  (* -------------------------------------------------------------
    Load-Error 							
  --------------------------------------------------------------*)
  JAM_ERROR                                 := 0180, // Jam Detected - Remove TU before restart 
  POSITION_OCCUPIED_AFTER_HANDOVER          := 0181, // Position occupied after transmission 
  POSITION_OCCUPIED_BEFORE_TAKEOVER         := 0182, // Position occupied before pickup 
  POSITION_NOT_CORRECT_OCCUPIED             := 0183, // Position is not correctly occupied 
  LOAD_CONTROL                              := 0184, // Check load for overhang 
  POSITION_LANE_FULL                        := 0185, // Position/Lane is full, remove some TU's 
  TRANSFER_ERROR                            := 0186, // Error during transfer
  LOAD_TOO_HIGH                             := 0187, // Load is too high
  LOAD_TOO_HEAVY                            := 0188, // Load is too heavy


  (* -------------------------------------------------------------
    Errors Drives						
  --------------------------------------------------------------*)
  DRIVE_ERROR                               := 0200, // Drive error 
  DRIVE_WARNING                             := 0201, // Drive warning 


  (*-------------------------------------------------------------
    Errors Scanners						
  --------------------------------------------------------------*)
  SCANNER_NO_READ                           := 0220, // Scanner could not read the label 
  SCANNER_CONTINOUS_NO_READ                 := 0221, // Continuous no reading 
  SCANNER_NO_DATA_RECEIVED                  := 0222, // No data received from scanner 
  SCANNER_NO_HANDSHAKE                      := 0223, // No handshake signal from scanner received 


  (* -------------------------------------------------------------
    Misc      
  --------------------------------------------------------------*)
  INIT_NOT_POSSIBLE                         := 0300, // Initialization was not possible
  START_NOT_POSSIBLE                        := 0301, // Starting not possible
  POSITIONING_ERROR                         := 0302, // Positioning error 
  INCORRECT_POSITION                        := 0303, // Actual position is not correct 
  BELT_BROKEN                               := 0304, // Belt is broken 
  DEVICE_ERROR                              := 0305, // Device error
  DEVICE_OFFLINE                            := 0306, // device is offline e.g. printer, scanner 
  WATCHDOG_ERROR                            := 0307, // Watchdog error 
  FILE_SYSTEM_ERROR                         := 0308, // Error during deleting file 
  DOOR_ERROR                                := 0309, // Maintenance door is open error 
  WRONG_MODE                                := 0310, // Manual mode is not active for performing manual movement 
  NOT_SUPPORTED                             := 0311, // Not supported message


  (* -------------------------------------------------------------
    Software errors       
  --------------------------------------------------------------*)
  CONFIGURATION_ERROR                       := 0900, // Configuration error 
  SOFTWARE_ERROR                            := 0901  // General software error 
);
END_TYPE

// ---- 20_Product/10_BCF/11_Conv/10_Base/01_DUTs/E_EtherCAT_MasterError.TcDUT
TYPE E_EtherCAT_MasterError :
(**************************************************************************************
 * 	Application		:	BoxControl Framework
 *	Revision		:	$Revision: 404529 $
 *	Revision date	:	$Date: 2018-04-23 08:21:38 +0200 (Mo., 23 Apr 2018) $
 *	Last changed by	:	$Author: b7bolm $
 *	URL				:	$URL: http://almscdc.swisslog.com/repo/SWPD/Development/BoxControlFramework/20_Release/trunk/01_Software/BCF/BCF/JumpStart/20_Product/10_App/10_Base/10_Lib/10_Conv/01_DUTs/E_EtherCAT_MasterError.TcDUT $
 *
 *	Purpose			:	EtherCAT master error
 *
 * ------------------------------------------------------------------------------------
 *	Copyright Swisslog [IP AG], Switzerland. All rights reserved.
 * 
 * ------------------------------------------------------------------------------------
 *	
 * 	Revision History: 
 *
 * 	VERSION			DATE			INITIALS			DESCRIPTION
 *	0.1				01.01.2001		swl					Example
 *
 **************************************************************************************)
(
	ETHERCAT_MASTER_NO_ERROR		:= 16#0000, // No error 
	LINK_ERROR 						:= 16#0001, // Link error  
	IO_LOCKED_AFTER_LINK_ERR		:= 16#0002, // I/O locked after link error (I/O reset required) 
	LINK_ERROR_REDUNDANCY_ADAPTER	:= 16#0004, // Link error (redundancy adapter) 
	MISSING_ONE_FRAME				:= 16#0008, // Missing one frame (redundancy mode) 
	OUT_OF_SEND_RESSOURCES			:= 16#0010, // Out OF send resources (I/O reset required) 
	WATCHDOG_TRIGGERED				:= 16#0020, // Watchdog triggered 
	ETHERNET_DRV_NOT_FOUND			:= 16#0040, // Ethernet driver (miniport) NOT found 
	IO_RESET_ACTIVE					:= 16#0080, // I/O reset active
	ONE_DEVICE_IN_INIT				:= 16#0100, // AT least one device in 'INIT' state 
	ONE_DEVICE_IN_PRE_OP			:= 16#0200, // AT least one device in 'PRE-OP' state 
	ONE_DEVICE_IN_SAFE_OP			:= 16#0400, // AT least one device in 'SAFE-OP' state 
	ONE_DEVICE_IN_ERROR				:= 16#0800, // AT least one device indicates an error state 
	DC_NOT_IN_SYNC					:= 16#1000  // DC NOT in sync 
);
END_TYPE

// ---- 20_Product/10_BCF/11_Conv/10_Base/01_DUTs/ST_ControlRequest.TcDUT
TYPE ST_ControlRequest :
(**************************************************************************************
 * 	Application		:	BoxControl Framework
 *	Revision		:	$Revision: 404529 $
 *	Revision date	:	$Date: 2018-04-23 08:21:38 +0200 (Mo., 23 Apr 2018) $
 *	Last changed by	:	$Author: b7bolm $
 *	URL				:	$URL: http://almscdc.swisslog.com/repo/SWPD/Development/BoxControlFramework/20_Release/trunk/01_Software/BCF/BCF/JumpStart/20_Product/10_App/10_Base/10_Lib/10_Conv/01_DUTs/ST_ControlRequest.TcDUT $
 *
 *	Purpose			:	Control request consists of a control code and value. These 
 *						values are normaly set by an ITC message.
 *
 * ------------------------------------------------------------------------------------
 *	Copyright Swisslog [IP AG], Switzerland. All rights reserved.
 * 
 * ------------------------------------------------------------------------------------
 *	
 * 	Revision History: 
 *
 * 	VERSION			DATE			INITIALS			DESCRIPTION
 *	0.1				01.01.2001		swl					Example
 *
 **************************************************************************************)
STRUCT
	ControlCode			: INT; // Control code from the control telegram 
	ControlValue		: INT; // Control value from the control telegram 
END_STRUCT
END_TYPE

// ---- 20_Product/10_BCF/11_Conv/10_Base/01_DUTs/ST_DataSet.TcDUT
TYPE ST_DataSet :
(**************************************************************************************
 * 	Application		:	BoxControl Framework
 *	Revision		:	$Revision: 411223 $
 *	Revision date	:	$Date: 2018-07-27 11:40:44 +0200 (Fr., 27 Jul 2018) $
 *	Last changed by	:	$Author: b7bolm $
 *	URL				:	$URL: http://almscdc.swisslog.com/repo/SWPD/Development/BoxControlFramework/20_Release/trunk/01_Software/BCF/BCF/JumpStart/20_Product/10_App/10_Base/10_Lib/10_Conv/01_DUTs/ST_DataSet.TcDUT $
 *
 *	Purpose			:	TU Data - Data set
 *
 * ------------------------------------------------------------------------------------
 *	Copyright Swisslog [IP AG], Switzerland. All rights reserved.
 * 
 * ------------------------------------------------------------------------------------
 *	
 * 	Revision History: 
 *
 * 	VERSION			DATE			INITIALS			DESCRIPTION
 *	0.1				01.01.2001		swl					Example
 *
 **************************************************************************************)
STRUCT
	DataPresent		: BOOL; // Data present 
	JobPresent		: BOOL; // Transfer order 
	TU_Type			: INT; // Type of transport unit 
	IO_Data			: INT; // Project specific data 
	Sequence		: ULINT; // 19 digit global sequence identifier
	SubSequence		: DINT; // 9 digit position in the sequence
	SequenceSize	: DINT; // 9 digit number of TU's in the sequence
	GroupID			: ULINT; // 19 digit global group identifier 
	GroupSize		: DINT; // 9 digit number of TU's in the group ID
	DestinationSlot	: INT; // 3 digit logical sub destination of destination
	NumberOfDest	: INT; // Number of destinations 
	Dimension		: ST_Dimension; // Dimensions
	Orientation		: STRING;	
	LowerLimit		: DINT; // Lower limit 
	UpperLimit		: DINT; // Upper limit
	TU_Parameter	: INT; // TU Parameter
	CheckpointID	: STRING(5); // Checkpoint ID
	HaltSequencing	: BOOL; // Sequencing information is temporally not valid
END_STRUCT
END_TYPE

// ---- 20_Product/10_BCF/11_Conv/10_Base/01_DUTs/ST_DataSetEmulation.TcDUT
TYPE ST_DataSetEmulation :
(**************************************************************************************
 * 	Application		:	BoxControl Framework
 *	Revision		:	$Revision: 404529 $
 *	Revision date	:	$Date: 2018-04-23 08:21:38 +0200 (Mo., 23 Apr 2018) $
 *	Last changed by	:	$Author: b7bolm $
 *	URL				:	$URL: http://almscdc.swisslog.com/repo/SWPD/Development/BoxControlFramework/20_Release/trunk/01_Software/BCF/BCF/JumpStart/20_Product/11_Emu/10_Base/10_Lib/10_Conv/01_DUTs/ST_DataSetEmulation.TcDUT $
 *
 *	Purpose			:	TU Data - Data set - Emulation
 *
 * ------------------------------------------------------------------------------------
 *	Copyright Swisslog [IP AG], Switzerland. All rights reserved.
 * 
 * ------------------------------------------------------------------------------------
 *	
 * 	Revision History: 
 *
 * 	VERSION			DATE			INITIALS			DESCRIPTION
 *	0.1				01.01.2001		swl					Example
 *
 **************************************************************************************)
STRUCT
	DataPresent		: BOOL; // Data present
	LongSideLeading : BOOL; // TU runs long side leading
	NestedIndex		: DINT; // Index of nested data set
	ParentIndex		: DINT; // Index of parent in view of nested
 	Dimension		: ST_Dimension; // Dimensions
END_STRUCT
END_TYPE

// ---- 20_Product/10_BCF/11_Conv/10_Base/01_DUTs/ST_Dimension.TcDUT
TYPE ST_Dimension :
(**************************************************************************************
 * 	Application		:	BoxControl Framework
 *	Revision		:	$Revision: 404529 $
 *	Revision date	:	$Date: 2018-04-23 08:21:38 +0200 (Mo., 23 Apr 2018) $
 *	Last changed by	:	$Author: b7bolm $
 *	URL				:	$URL: http://almscdc.swisslog.com/repo/SWPD/Development/BoxControlFramework/20_Release/trunk/01_Software/BCF/BCF/JumpStart/20_Product/10_App/10_Base/10_Lib/10_Conv/01_DUTs/ST_Dimension.TcDUT $
 *
 *	Purpose			:	TU Data - Dimension
 *
 * ------------------------------------------------------------------------------------
 *	Copyright Swisslog [IP AG], Switzerland. All rights reserved.
 * 
 * ------------------------------------------------------------------------------------
 *	
 * 	Revision History: 
 *
 * 	VERSION			DATE			INITIALS			DESCRIPTION
 *	0.1				01.01.2001		swl					Example
 *
 **************************************************************************************)
STRUCT
	Length		: INT; // Length
	Width		: INT; // Width
	Height		: INT; // Height
	Weight		: DINT; // Weight
END_STRUCT
END_TYPE

// ---- 20_Product/10_BCF/11_Conv/10_Base/01_DUTs/ST_ElementRegistryConv.TcDUT
TYPE ST_ElementRegistryConv :
(**************************************************************************************
 * 	Application		:	BoxControl Framework
 *	Revision		:	$Revision: 404529 $
 *	Revision date	:	$Date: 2018-04-23 08:21:38 +0200 (Mo., 23 Apr 2018) $
 *	Last changed by	:	$Author: b7bolm $
 *	URL				:	$URL: http://almscdc.swisslog.com/repo/SWPD/Development/BoxControlFramework/20_Release/trunk/01_Software/BCF/BCF/JumpStart/20_Product/10_App/10_Base/10_Lib/10_Conv/01_DUTs/ST_ElementRegistryConv.TcDUT $
 *
 *	Purpose			:	Element registration structure.
 *
 * ------------------------------------------------------------------------------------
 *	Copyright Swisslog [IP AG], Switzerland. All rights reserved.
 * 
 * ------------------------------------------------------------------------------------
 *	
 * 	Revision History: 
 *
 * 	VERSION			DATE			INITIALS			DESCRIPTION
 *	0.1				01.01.2001		swl					Example
 *
 **************************************************************************************)
STRUCT
	Enable				: BOOL; // Element enabled 
	ElementName			: STRING(System.NAME_LENGTH); // Name as string
	eElementNumber		: E_ElementNumber; // Element number 
	eElementType		: E_ElementType; // Element type
	rElementData		: REFERENCE TO ST_ElementData; 
	rElementInterface 	: REFERENCE TO ST_ElementInterface;
	rSettingsElement	: REFERENCE TO ST_CFG_Element;
	rElement			: REFERENCE TO FB_ElementConv; // Reference to Element 
	HashCode			: UDINT; // HashCode
END_STRUCT
END_TYPE

// ---- 20_Product/10_BCF/11_Conv/10_Base/01_DUTs/ST_ElementRegistryConvEmulation.TcDUT
TYPE ST_ElementRegistryConvEmulation :
(**************************************************************************************
 * 	Application		:	BoxControl Framework
 *	Revision		:	$Revision: 404529 $
 *	Revision date	:	$Date: 2018-04-23 08:21:38 +0200 (Mo., 23 Apr 2018) $
 *	Last changed by	:	$Author: b7bolm $
 *	URL				:	$URL: http://almscdc.swisslog.com/repo/SWPD/Development/BoxControlFramework/20_Release/trunk/01_Software/BCF/BCF/JumpStart/20_Product/11_Emu/10_Base/10_Lib/10_Conv/01_DUTs/ST_ElementRegistryConvEmulation.TcDUT $
 *
 *	Purpose			:	Element registration structure - Emulation.
 *
 * ------------------------------------------------------------------------------------
 *	Copyright Swisslog [IP AG], Switzerland. All rights reserved.
 * 
 * ------------------------------------------------------------------------------------
 *	
 * 	Revision History: 
 *
 * 	VERSION			DATE			INITIALS			DESCRIPTION
 *	0.1				01.01.2001		swl					Example
 *
 **************************************************************************************)
STRUCT
	rElement			: REFERENCE TO FB_ElementConvEmulation; // Element object reference
END_STRUCT
END_TYPE

// ---- 20_Product/10_BCF/11_Conv/10_Base/01_DUTs/ST_ErrorDataSet.TcDUT
TYPE ST_ErrorDataSet :
(**************************************************************************************
 * 	Application		:	BoxControl Framework
 *	Revision		:	$Revision: 404529 $
 *	Revision date	:	$Date: 2018-04-23 08:21:38 +0200 (Mo., 23 Apr 2018) $
 *	Last changed by	:	$Author: b7bolm $
 *	URL				:	$URL: http://almscdc.swisslog.com/repo/SWPD/Development/BoxControlFramework/20_Release/trunk/01_Software/BCF/BCF/JumpStart/20_Product/10_App/10_Base/10_Lib/10_Conv/01_DUTs/ST_ErrorDataSet.TcDUT $
 *
 *	Purpose			:	Error data set
 *
 * ------------------------------------------------------------------------------------
 *	Copyright Swisslog [IP AG], Switzerland. All rights reserved.
 * 
 * ------------------------------------------------------------------------------------
 *	
 * 	Revision History: 
 *
 * 	VERSION			DATE			INITIALS			DESCRIPTION
 *	0.1				01.01.2001		swl					Example
 *
 **************************************************************************************)
STRUCT
	ErrorType		: E_ErrorType;	// Type of error 
	ErrorCode		: U_ErrorCode; // Type casting for error code by product or framework errors 
	ErrorParam		: STRING(System.ERROR_PARAM_STRINGLENGTH); // Error parameter 
	ResetError		: BOOL; // Command to reset error 
END_STRUCT
END_TYPE

// ---- 20_Product/10_BCF/11_Conv/10_Base/01_DUTs/ST_EtherCATDeviceStates.TcDUT
TYPE ST_EtherCATDeviceStates :
(**************************************************************************************
 * 	Application		:	BoxControl Framework
 *	Revision		:	$Revision: 404529 $
 *	Revision date	:	$Date: 2018-04-23 08:21:38 +0200 (Mo., 23 Apr 2018) $
 *	Last changed by	:	$Author: b7bolm $
 *	URL				:	$URL: http://almscdc.swisslog.com/repo/SWPD/Development/BoxControlFramework/20_Release/trunk/01_Software/BCF/BCF/JumpStart/20_Product/10_App/10_Base/10_Lib/10_Conv/01_DUTs/ST_EtherCATDeviceStates.TcDUT $
 *
 *	Purpose			:	Supervision of EtherCAT slaves.
 *
 * ------------------------------------------------------------------------------------
 *	Copyright Swisslog [IP AG], Switzerland. All rights reserved.
 * 
 * ------------------------------------------------------------------------------------
 *	
 * 	Revision History: 
 *
 * 	VERSION			DATE			INITIALS			DESCRIPTION
 *	0.1				01.01.2001		swl					Example
 *
 **************************************************************************************)
STRUCT
	LastDeviceState	  	: UINT; // Last device states
	DeviceState	 		: UINT; // Current device state
	EventDateTime		: DATE_AND_TIME; // Event time of last error
	Error				: BOOL; // Error active
END_STRUCT
END_TYPE

// ---- 20_Product/10_BCF/11_Conv/10_Base/01_DUTs/ST_ExecutionTime.TcDUT
TYPE ST_ExecutionTime :
(**************************************************************************************
 * 	Application		:	BoxControl Framework
 *	Revision		:	$Revision: 404529 $
 *	Revision date	:	$Date: 2018-04-23 08:21:38 +0200 (Mo., 23 Apr 2018) $
 *	Last changed by	:	$Author: b7bolm $
 *	URL				:	$URL: http://almscdc.swisslog.com/repo/SWPD/Development/BoxControlFramework/20_Release/trunk/01_Software/BCF/BCF/JumpStart/20_Product/10_App/10_Base/10_Lib/10_Conv/01_DUTs/ST_ExecutionTime.TcDUT $
 *
 *	Purpose			:	Execution time
 *
 * ------------------------------------------------------------------------------------
 *	Copyright Swisslog [IP AG], Switzerland. All rights reserved.
 * 
 * ------------------------------------------------------------------------------------
 *	
 * 	Revision History: 
 *
 * 	VERSION			DATE			INITIALS			DESCRIPTION
 *	0.1				01.01.2001		swl					Example
 *
 **************************************************************************************)
STRUCT
	CurrentValue	: ULINT;
	MaxValue		: ULINT;
END_STRUCT
END_TYPE

// ---- 20_Product/10_BCF/11_Conv/10_Base/01_DUTs/ST_ExternalDestination.TcDUT
TYPE ST_ExternalDestination :
(**************************************************************************************
 * 	Application		:	BoxControl Framework
 *	Revision		:	$Revision: 404529 $
 *	Revision date	:	$Date: 2018-04-23 08:21:38 +0200 (Mo., 23 Apr 2018) $
 *	Last changed by	:	$Author: b7bolm $
 *	URL				:	$URL: http://almscdc.swisslog.com/repo/SWPD/Development/BoxControlFramework/20_Release/trunk/01_Software/BCF/BCF/JumpStart/20_Product/10_App/10_Base/10_Lib/10_Conv/01_DUTs/ST_ExternalDestination.TcDUT $
 *
 *	Purpose			:	External destination definition.
 *
 * ------------------------------------------------------------------------------------
 *	Copyright Swisslog [IP AG], Switzerland. All rights reserved.
 * 
 * ------------------------------------------------------------------------------------
 *	
 * 	Revision History: 
 *
 * 	VERSION			DATE			INITIALS			DESCRIPTION
 *	0.1				01.01.2001		swl					Example
 *
 **************************************************************************************)
STRUCT
	PositionName		: STRING(NAME_LENGTH);
	HashCode			: UDINT; // HashCode
END_STRUCT
END_TYPE

// ---- 20_Product/10_BCF/11_Conv/10_Base/01_DUTs/ST_FunctionRegistryConv.TcDUT
TYPE ST_FunctionRegistryConv :
(**************************************************************************************
 * 	Application		:	BoxControl Framework
 *	Revision		:	$Revision: 404529 $
 *	Revision date	:	$Date: 2018-04-23 08:21:38 +0200 (Mo., 23 Apr 2018) $
 *	Last changed by	:	$Author: b7bolm $
 *	URL				:	$URL: http://almscdc.swisslog.com/repo/SWPD/Development/BoxControlFramework/20_Release/trunk/01_Software/BCF/BCF/JumpStart/20_Product/10_App/10_Base/10_Lib/10_Conv/01_DUTs/ST_FunctionRegistryConv.TcDUT $
 *
 *	Purpose			:	Element function registration structure.
 *
 * ------------------------------------------------------------------------------------
 *	Copyright Swisslog [IP AG], Switzerland. All rights reserved.
 * 
 * ------------------------------------------------------------------------------------
 *	
 * 	Revision History: 
 *
 * 	VERSION			DATE			INITIALS			DESCRIPTION
 *	0.1				01.01.2001		swl					Example
 *
 **************************************************************************************)
STRUCT
	Enable					: BOOL; // Registry slot gets called
	FunctionName			: STRING(System.NAME_LENGTH); // Name as string
	eFunctionNumber			: E_FunctionNumber; // Identifier used as registration number
	eFunctionType			: E_FunctionType; // Type
	rFunctionData			: REFERENCE TO ST_FunctionData;
	rFunctionInterface		: REFERENCE TO ST_FunctionInterface;
	rSettingsFunction		: REFERENCE TO ST_CFG_Function;
	rFunction				: REFERENCE TO FB_FunctionConv; // Reference to function
	Zone					: ARRAY[1..Conveyor.NUMBER_OF_ZONES_PER_FUNCTION] OF ST_ZoneRegistryConv; // Zone registration values
	HashCode				: UDINT; // HashCode
END_STRUCT
END_TYPE

// ---- 20_Product/10_BCF/11_Conv/10_Base/01_DUTs/ST_FunctionRegistryConvEmulation.TcDUT
TYPE ST_FunctionRegistryConvEmulation :
(**************************************************************************************
 * 	Application		:	BoxControl Framework
 *	Revision		:	$Revision: 404529 $
 *	Revision date	:	$Date: 2018-04-23 08:21:38 +0200 (Mo., 23 Apr 2018) $
 *	Last changed by	:	$Author: b7bolm $
 *	URL				:	$URL: http://almscdc.swisslog.com/repo/SWPD/Development/BoxControlFramework/20_Release/trunk/01_Software/BCF/BCF/JumpStart/20_Product/11_Emu/10_Base/10_Lib/10_Conv/01_DUTs/ST_FunctionRegistryConvEmulation.TcDUT $
 *
 *	Purpose			:	Function registration structure - Emulation.
 *
 * ------------------------------------------------------------------------------------
 *	Copyright Swisslog [IP AG], Switzerland. All rights reserved.
 * 
 * ------------------------------------------------------------------------------------
 *	
 * 	Revision History: 
 *
 * 	VERSION			DATE			INITIALS			DESCRIPTION
 *	0.1				01.01.2001		swl					Example
 *
 **************************************************************************************)
STRUCT
	rFunction			: REFERENCE TO FB_FunctionConvEmulation; // Function object reference
END_STRUCT
END_TYPE

// ---- 20_Product/10_BCF/11_Conv/10_Base/01_DUTs/ST_GroupRegistryConv.TcDUT
TYPE ST_GroupRegistryConv :
(**************************************************************************************
 * 	Application		:	BoxControl Framework
 *	Revision		:	$Revision: 404529 $
 *	Revision date	:	$Date: 2018-04-23 08:21:38 +0200 (Mo., 23 Apr 2018) $
 *	Last changed by	:	$Author: b7bolm $
 *	URL				:	$URL: http://almscdc.swisslog.com/repo/SWPD/Development/BoxControlFramework/20_Release/trunk/01_Software/BCF/BCF/JumpStart/20_Product/10_App/10_Base/10_Lib/10_Conv/01_DUTs/ST_GroupRegistryConv.TcDUT $
 *
 *	Purpose			:	Group registration structure.
 *
 * ------------------------------------------------------------------------------------
 *	Copyright Swisslog [IP AG], Switzerland. All rights reserved.
 * 
 * ------------------------------------------------------------------------------------
 *	
 * 	Revision History: 
 *
 * 	VERSION			DATE			INITIALS			DESCRIPTION
 *	0.1				01.01.2001		swl					Example
 *
 **************************************************************************************)
STRUCT
	Enable				: BOOL; // Group call enabled
	GroupName			: STRING(System.NAME_LENGTH); // Name as string
	eGroupNumber		: E_GroupNumber; // Group enumeration number
	eGroupType			: E_GroupType; // Group type
	rGroupData			: REFERENCE TO ST_GroupData;
	rGroupInterface		: REFERENCE TO ST_GroupInterface;
	rSettingsGroup		: REFERENCE TO ST_CFG_Group;
	rGroup				: REFERENCE TO FB_GroupConv; // Group object reference
	HashCode			: UDINT; // HashCode
END_STRUCT
END_TYPE

// ---- 20_Product/10_BCF/11_Conv/10_Base/01_DUTs/ST_GroupRegistryConvEmulation.TcDUT
TYPE ST_GroupRegistryConvEmulation :
(**************************************************************************************
 * 	Application		:	BoxControl Framework
 *	Revision		:	$Revision: 404529 $
 *	Revision date	:	$Date: 2018-04-23 08:21:38 +0200 (Mo., 23 Apr 2018) $
 *	Last changed by	:	$Author: b7bolm $
 *	URL				:	$URL: http://almscdc.swisslog.com/repo/SWPD/Development/BoxControlFramework/20_Release/trunk/01_Software/BCF/BCF/JumpStart/20_Product/11_Emu/10_Base/10_Lib/10_Conv/01_DUTs/ST_GroupRegistryConvEmulation.TcDUT $
 *
 *	Purpose			:	Group registration structure - Emulation.
 *
 * ------------------------------------------------------------------------------------
 *	Copyright Swisslog [IP AG], Switzerland. All rights reserved.
 * 
 * ------------------------------------------------------------------------------------
 *	
 * 	Revision History: 
 *
 * 	VERSION			DATE			INITIALS			DESCRIPTION
 *	0.1				01.01.2001		swl					Example
 *
 **************************************************************************************)
STRUCT
	rGroup			: REFERENCE TO FB_GroupConvEmulation; // Group object reference
END_STRUCT
END_TYPE

// ---- 20_Product/10_BCF/11_Conv/10_Base/01_DUTs/ST_InitRelease.TcDUT
TYPE ST_InitRelease :
(**************************************************************************************
 * 	Application		:	BoxControl Framework
 *	Revision		:	$Revision: 404529 $
 *	Revision date	:	$Date: 2018-04-23 08:21:38 +0200 (Mo., 23 Apr 2018) $
 *	Last changed by	:	$Author: b7bolm $
 *	URL				:	$URL: http://almscdc.swisslog.com/repo/SWPD/Development/BoxControlFramework/20_Release/trunk/01_Software/BCF/BCF/JumpStart/20_Product/10_App/10_Base/10_Lib/10_Conv/01_DUTs/ST_InitRelease.TcDUT $
 *
 *	Purpose			:	 Init release
 *
 * ------------------------------------------------------------------------------------
 *	Copyright Swisslog [IP AG], Switzerland. All rights reserved.
 * 
 * ------------------------------------------------------------------------------------
 *	
 * 	Revision History: 
 *
 * 	VERSION			DATE			INITIALS			DESCRIPTION
 *	0.1				01.01.2001		swl					Example
 *
 **************************************************************************************)
STRUCT
	eLimitFunctionNumber	: E_FunctionNumber;
	eLimitElementNumber		: E_ElementNumber;
	eLimitGroup				: E_GroupNumber;
END_STRUCT
END_TYPE

// ---- 20_Product/10_BCF/11_Conv/10_Base/01_DUTs/ST_Interlock.TcDUT
TYPE ST_Interlock :
(**************************************************************************************
 * 	Application		:	BoxControl Framework
 *	Revision		:	$Revision: 404529 $
 *	Revision date	:	$Date: 2018-04-23 08:21:38 +0200 (Mo., 23 Apr 2018) $
 *	Last changed by	:	$Author: b7bolm $
 *	URL				:	$URL: http://almscdc.swisslog.com/repo/SWPD/Development/BoxControlFramework/20_Release/trunk/01_Software/BCF/BCF/JumpStart/20_Product/10_App/10_Base/10_Lib/10_Conv/01_DUTs/ST_Interlock.TcDUT $
 *
 *	Purpose			:	General interlock structure
 *
 * ------------------------------------------------------------------------------------
 *	Copyright Swisslog [IP AG], Switzerland. All rights reserved.
 * 
 * ------------------------------------------------------------------------------------
 *	
 * 	Revision History: 
 *
 * 	VERSION			DATE			INITIALS			DESCRIPTION
 *	0.1				01.01.2001		swl					Example
 *
 **************************************************************************************)
STRUCT
	Enable			: BOOL;
	Stop			: BOOL;
	ConveyEnable	: BOOL;
END_STRUCT
END_TYPE

// ---- 20_Product/10_BCF/11_Conv/10_Base/01_DUTs/ST_Label.TcDUT
TYPE ST_Label :
(**************************************************************************************
 * 	Application		:	BoxControl Framework
 *	Revision		:	$Revision: 404529 $
 *	Revision date	:	$Date: 2018-04-23 08:21:38 +0200 (Mo., 23 Apr 2018) $
 *	Last changed by	:	$Author: b7bolm $
 *	URL				:	$URL: http://almscdc.swisslog.com/repo/SWPD/Development/BoxControlFramework/20_Release/trunk/01_Software/BCF/BCF/JumpStart/20_Product/10_App/10_Base/10_Lib/10_Conv/01_DUTs/ST_Label.TcDUT $
 *
 *	Purpose			:	TU Data - Label
 *
 * ------------------------------------------------------------------------------------
 *	Copyright Swisslog [IP AG], Switzerland. All rights reserved.
 * 
 * ------------------------------------------------------------------------------------
 *	
 * 	Revision History: 
 *
 * 	VERSION			DATE			INITIALS			DESCRIPTION
 *	0.1				01.01.2001		swl					Example
 *
 **************************************************************************************)
STRUCT
	ASCII		: STRING(Conveyor.LABEL_LENGTH); // Label
END_STRUCT
END_TYPE

// ---- 20_Product/10_BCF/11_Conv/10_Base/01_DUTs/ST_LabelEmulation.TcDUT
TYPE ST_LabelEmulation :
(**************************************************************************************
 * 	Application		:	BoxControl Framework
 *	Revision		:	$Revision: 404529 $
 *	Revision date	:	$Date: 2018-04-23 08:21:38 +0200 (Mo., 23 Apr 2018) $
 *	Last changed by	:	$Author: b7bolm $
 *	URL				:	$URL: http://almscdc.swisslog.com/repo/SWPD/Development/BoxControlFramework/20_Release/trunk/01_Software/BCF/BCF/JumpStart/20_Product/11_Emu/10_Base/10_Lib/10_Conv/01_DUTs/ST_LabelEmulation.TcDUT $
 *
 *	Purpose			:	Emulation label
 *
 * ------------------------------------------------------------------------------------
 *	Copyright Swisslog [IP AG], Switzerland. All rights reserved.
 * 
 * ------------------------------------------------------------------------------------
 *	
 * 	Revision History: 
 *
 * 	VERSION			DATE			INITIALS			DESCRIPTION
 *	0.1				01.01.2001		swl					Example
 *
 **************************************************************************************)
STRUCT
	ASCII		: STRING(Conveyor.LABEL_LENGTH); // Label
	HashCode	: UDINT; // Hashcode
END_STRUCT
END_TYPE

// ---- 20_Product/10_BCF/11_Conv/10_Base/01_DUTs/ST_PositionIdent.TcDUT
TYPE ST_PositionIdent :
(**************************************************************************************
 * 	Application		:	BoxControl Framework
 *	Revision		:	$Revision: 404529 $
 *	Revision date	:	$Date: 2018-04-23 08:21:38 +0200 (Mo., 23 Apr 2018) $
 *	Last changed by	:	$Author: b7bolm $
 *	URL				:	$URL: http://almscdc.swisslog.com/repo/SWPD/Development/BoxControlFramework/20_Release/trunk/01_Software/BCF/BCF/JumpStart/20_Product/10_App/10_Base/10_Lib/10_Conv/01_DUTs/ST_PositionIdent.TcDUT $
 *
 *	Purpose			:	Position identification.
 *
 * ------------------------------------------------------------------------------------
 *	Copyright Swisslog [IP AG], Switzerland. All rights reserved.
 * 
 * ------------------------------------------------------------------------------------
 *	
 * 	Revision History: 
 *
 * 	VERSION			DATE			INITIALS			DESCRIPTION
 *	0.1				01.01.2001		swl					Example
 *
 **************************************************************************************)
STRUCT
	eFunctionNumber		: E_FunctionNumber; // Number of the function
	ZoneNumber			: INT; // Number of the zone in the function
	PositionName		: STRING(NAME_LENGTH);
END_STRUCT
END_TYPE

// ---- 20_Product/10_BCF/11_Conv/10_Base/01_DUTs/ST_Profile.TcDUT
TYPE ST_Profile :
(**************************************************************************************
 * 	Application		:	BoxControl Framework
 *	Revision		:	$Revision: 404529 $
 *	Revision date	:	$Date: 2018-04-23 08:21:38 +0200 (Mo., 23 Apr 2018) $
 *	Last changed by	:	$Author: b7bolm $
 *	URL				:	$URL: http://almscdc.swisslog.com/repo/SWPD/Development/BoxControlFramework/20_Release/trunk/01_Software/BCF/BCF/JumpStart/20_Product/10_App/10_Base/10_Lib/10_Conv/01_DUTs/ST_Profile.TcDUT $
 *
 *	Purpose			:	TU Data - Profile
 *
 * ------------------------------------------------------------------------------------
 *	Copyright Swisslog [IP AG], Switzerland. All rights reserved.
 * 
 * ------------------------------------------------------------------------------------
 *	
 * 	Revision History: 
 *
 * 	VERSION			DATE			INITIALS			DESCRIPTION
 *	0.1				01.01.2001		swl					Example
 *
 **************************************************************************************)
STRUCT
	Height			: INT; // Height 
	ProfileLeft		: INT; // Profile left 
	ProfileRight	: INT; // Profile right 
	ProfileFront	: INT; // Profile front 
	ProfileRear		: INT; // Profile rear
	Tunnel			: INT; // Tunnel 
	Runner			: INT; // Runner 
	Weight			: DINT; // Weight 
END_STRUCT
END_TYPE

// ---- 20_Product/10_BCF/11_Conv/10_Base/01_DUTs/ST_SubSystemRegistryConv.TcDUT
TYPE ST_SubSystemRegistryConv :
(**************************************************************************************
 * 	Application		:	BoxControl Framework
 *	Revision		:	$Revision: 404529 $
 *	Revision date	:	$Date: 2018-04-23 08:21:38 +0200 (Mo., 23 Apr 2018) $
 *	Last changed by	:	$Author: b7bolm $
 *	URL				:	$URL: http://almscdc.swisslog.com/repo/SWPD/Development/BoxControlFramework/20_Release/trunk/01_Software/BCF/BCF/JumpStart/20_Product/10_App/10_Base/10_Lib/10_Conv/01_DUTs/ST_SubSystemRegistryConv.TcDUT $
 *
 *	Purpose			:	Subsystem registration structure.
 *
 * ------------------------------------------------------------------------------------
 *	Copyright Swisslog [IP AG], Switzerland. All rights reserved.
 * 
 * ------------------------------------------------------------------------------------
 *	
 * 	Revision History: 
 *
 * 	VERSION			DATE			INITIALS			DESCRIPTION
 *	0.1				01.01.2001		swl					Example
 *
 **************************************************************************************)
STRUCT
	SubsystemName			: STRING(System.NAME_LENGTH); // Name as string
	rSubsystemData			: REFERENCE TO ST_SubsystemData;
	rSubsystemInterface 	: REFERENCE TO ST_SubsystemInterface;
	rSettingsSubsystem	 	: REFERENCE TO ST_CFG_Subsystem;
	rSubsystem				: REFERENCE TO FB_SubsystemConv;
	HashCode				: UDINT; // HashCode
END_STRUCT
END_TYPE

// ---- 20_Product/10_BCF/11_Conv/10_Base/01_DUTs/ST_SubsystemRegistryConvEmulation.TcDUT
TYPE ST_SubsystemRegistryConvEmulation :
(**************************************************************************************
 * 	Application		:	BoxControl Framework
 *	Revision		:	$Revision: 404529 $
 *	Revision date	:	$Date: 2018-04-23 08:21:38 +0200 (Mo., 23 Apr 2018) $
 *	Last changed by	:	$Author: b7bolm $
 *	URL				:	$URL: http://almscdc.swisslog.com/repo/SWPD/Development/BoxControlFramework/20_Release/trunk/01_Software/BCF/BCF/JumpStart/20_Product/11_Emu/10_Base/10_Lib/10_Conv/01_DUTs/ST_SubsystemRegistryConvEmulation.TcDUT $
 *
 *	Purpose			:	Subsystem registration structure - Emulation.
 *
 * ------------------------------------------------------------------------------------
 *	Copyright Swisslog [IP AG], Switzerland. All rights reserved.
 * 
 * ------------------------------------------------------------------------------------
 *	
 * 	Revision History: 
 *
 * 	VERSION			DATE			INITIALS			DESCRIPTION
 *	0.1				01.01.2001		swl					Example
 *
 **************************************************************************************)
STRUCT
	rSubsystem			: REFERENCE TO FB_SubsystemConvEmulation; // Subsystem object reference
END_STRUCT
END_TYPE

// ---- 20_Product/10_BCF/11_Conv/10_Base/01_DUTs/ST_TimeStamp.TcDUT
TYPE ST_TimeStamp :
(**************************************************************************************
 * 	Application		:	BoxControl Framework
 *	Revision		:	$Revision: 404529 $
 *	Revision date	:	$Date: 2018-04-23 08:21:38 +0200 (Mo., 23 Apr 2018) $
 *	Last changed by	:	$Author: b7bolm $
 *	URL				:	$URL: http://almscdc.swisslog.com/repo/SWPD/Development/BoxControlFramework/20_Release/trunk/01_Software/BCF/BCF/JumpStart/20_Product/10_App/10_Base/10_Lib/10_Conv/01_DUTs/ST_TimeStamp.TcDUT $
 *
 *	Purpose			:	TU Data Time Stamp
 *
 * ------------------------------------------------------------------------------------
 *	Copyright Swisslog [IP AG], Switzerland. All rights reserved.
 * 
 * ------------------------------------------------------------------------------------
 *	
 * 	Revision History: 
 *
 * VERSION DATE         INITIALS     DESCRIPTION
 * 0.0     DD.MM.YYYY   (name)       (explain customized modifications)
 *
 **************************************************************************************)
STRUCT
	eInsertFunctionNumber		: E_FunctionNumber			:= 0;	// Inserted function number
	InsertZoneNumber			: INT						:= 0;	// Inserted zone number
	InsertDateTime				: Tc2_Utilities.TIMESTRUCT;			// Date and time of the insert 
END_STRUCT
END_TYPE

// ---- 20_Product/10_BCF/11_Conv/10_Base/01_DUTs/ST_TU_Data.TcDUT
TYPE ST_TU_Data :
(**************************************************************************************
 * 	Application		:	BoxControl Framework
 *	Revision		:	$Revision: 465877 $
 *	Revision date	:	$Date: 2020-11-17 14:28:17 +0100 (tis, 17 nov 2020) $
 *	Last changed by	:	$Author: b7lipim $
 *	URL				:	$URL: http://almscdc.swisslog.com/repo/SWPD/Development/BoxControlFramework/20_Release/tags/R1.12.0/01_Software/BCF/BCF/JumpStart/20_Product/10_BCF/11_Conv/10_Base/01_DUTs/ST_TU_Data.TcDUT $
 *
 *	Purpose			:	TU Data
 *
 * ------------------------------------------------------------------------------------
 *	Copyright Swisslog [IP AG], Switzerland. All rights reserved.
 * 
 * ------------------------------------------------------------------------------------
 *	
 * 	Revision History: 
 *
 * VERSION DATE         INITIALS     DESCRIPTION
 * 0.0     DD.MM.YYYY   (name)       (explain customized modifications)
 *
 **************************************************************************************)
STRUCT
  DataSet               : ST_DataSet; // DataSet 
  TU_ID                 : ST_TU_ID; // TU-ID 
  AssignmentID          : UDINT; // Assignment ID
  Label                 : ST_Label; // Label 
  Destination           : ARRAY[1..NUMBER_OF_DESTINATIONS] OF ST_PositionIdent; // PositionNumber and index 
  Profile               : ST_Profile; // Profile
  TimeStamp             : ST_TimeStamp; // TimeStamp 
  CurrentFunctionNumber : E_FunctionNumber; // Current function where the TU is located
  CurrentZoneNumber     : INT; // Current zone where the TU is located
END_STRUCT
END_TYPE

// ---- 20_Product/10_BCF/11_Conv/10_Base/01_DUTs/ST_TU_DataEmulation.TcDUT
TYPE ST_TU_DataEmulation :
(**************************************************************************************
 * 	Application		:	BoxControl Framework
 *	Revision		:	$Revision: 412414 $
 *	Revision date	:	$Date: 2018-08-17 07:57:24 +0200 (Fr., 17 Aug 2018) $
 *	Last changed by	:	$Author: d7herza $
 *	URL				:	$URL: http://almscdc.swisslog.com/repo/SWPD/Development/BoxControlFramework/20_Release/trunk/01_Software/BCF/BCF/JumpStart/20_Product/11_Emu/10_Base/10_Lib/10_Conv/01_DUTs/ST_TU_DataEmulation.TcDUT $
 *
 *	Purpose			:	TU Data
 *
 * ------------------------------------------------------------------------------------
 *	Copyright Swisslog [IP AG], Switzerland. All rights reserved.
 * 
 * ------------------------------------------------------------------------------------
 *	
 * 	Revision History: 
 *
 * 	VERSION			DATE			INITIALS			DESCRIPTION
 *	0.1				01.01.2001		swl					Example
 *
 **************************************************************************************)
STRUCT
	DataSet			: ST_DataSetEmulation; // DataSet
	Label			: ST_LabelEmulation; // Label
	TimeStamp		: ST_TimeStamp; // TimeStamp 
END_STRUCT
END_TYPE

// ---- 20_Product/10_BCF/11_Conv/10_Base/01_DUTs/ST_TU_ID.TcDUT
TYPE ST_TU_ID :
(**************************************************************************************
 * 	Application		:	BoxControl Framework
 *	Revision		:	$Revision: 404529 $
 *	Revision date	:	$Date: 2018-04-23 08:21:38 +0200 (Mo., 23 Apr 2018) $
 *	Last changed by	:	$Author: b7bolm $
 *	URL				:	$URL: http://almscdc.swisslog.com/repo/SWPD/Development/BoxControlFramework/20_Release/trunk/01_Software/BCF/BCF/JumpStart/20_Product/10_App/10_Base/10_Lib/10_Conv/01_DUTs/ST_TU_ID.TcDUT $
 *
 *	Purpose			:	TU ID
 *
 * ------------------------------------------------------------------------------------
 *	Copyright Swisslog [IP AG], Switzerland. All rights reserved.
 * 
 * ------------------------------------------------------------------------------------
 *	
 * 	Revision History: 
 *
 * 	VERSION			DATE			INITIALS			DESCRIPTION
 *	0.1				01.01.2001		swl					Example
 *
 **************************************************************************************)
STRUCT
	ASCII		: STRING(Conveyor.TU_ID_STRINGLENGTH); // TU_ID as characters 1 to 18 
	HashCode	: UDINT; // HashCode 
END_STRUCT
END_TYPE

// ---- 20_Product/10_BCF/11_Conv/10_Base/01_DUTs/ST_ZoneRegistryConv.TcDUT
TYPE ST_ZoneRegistryConv :
(**************************************************************************************
 * 	Application		:	BoxControl Framework
 *	Revision		:	$Revision: 404529 $
 *	Revision date	:	$Date: 2018-04-23 08:21:38 +0200 (Mo., 23 Apr 2018) $
 *	Last changed by	:	$Author: b7bolm $
 *	URL				:	$URL: http://almscdc.swisslog.com/repo/SWPD/Development/BoxControlFramework/20_Release/trunk/01_Software/BCF/BCF/JumpStart/20_Product/10_App/10_Base/10_Lib/10_Conv/01_DUTs/ST_ZoneRegistryConv.TcDUT $
 *
 *	Purpose			:	Zone registration structure.
 *
 * ------------------------------------------------------------------------------------
 *	Copyright Swisslog [IP AG], Switzerland. All rights reserved.
 * 
 * ------------------------------------------------------------------------------------
 *	
 * 	Revision History: 
 *
 * 	VERSION			DATE			INITIALS			DESCRIPTION
 *	0.1				01.01.2001		swl					Example
 *
 **************************************************************************************)
STRUCT
	ZoneName			: STRING(System.NAME_LENGTH); // Name as string
	refZoneData			: REFERENCE TO ST_ZoneData; // Internal function data
	refZoneInterface	: REFERENCE TO ST_ZoneInterface; // Function interface data
	HashCode			: UDINT; // HashCode
END_STRUCT
END_TYPE

// ---- 20_Product/10_BCF/11_Conv/10_Base/01_DUTs/U_ErrorCode.TcDUT
TYPE U_ErrorCode :
(**************************************************************************************
 * 	Application		:	BoxControl Framework
 *	Revision		:	$Revision: 404529 $
 *	Revision date	:	$Date: 2018-04-23 08:21:38 +0200 (Mo., 23 Apr 2018) $
 *	Last changed by	:	$Author: b7bolm $
 *	URL				:	$URL: http://almscdc.swisslog.com/repo/SWPD/Development/BoxControlFramework/20_Release/trunk/01_Software/BCF/BCF/JumpStart/20_Product/10_App/10_Base/10_Lib/10_Conv/01_DUTs/U_ErrorCode.TcDUT $
 *
 *	Purpose			:	Error list 
 *						All codes have to be set to a value!
 *
 * ------------------------------------------------------------------------------------
 *	Copyright Swisslog [IP AG], Switzerland. All rights reserved.
 * 
 * ------------------------------------------------------------------------------------
 *	
 * 	Revision History: 
 *
 * 	VERSION			DATE			INITIALS			DESCRIPTION
 *	0.1				01.01.2001		swl					Example
 *
 *************************************************************************************)	
UNION
	Conv	 	: E_ErrorConv; // Error BCF
	Product 	: E_ErrorProduct;  // Error product 
END_UNION
END_TYPE

// ---- 20_Product/10_BCF/11_Conv/10_Base/13_GroupManager/01_DUTs/ST_CFG_GroupManager.TcDUT
TYPE ST_CFG_GroupManager :
(**************************************************************************************
 * 	Application		:	Framework
 *	Revision		:	$Revision: 404529 $
 *	Revision date	:	$Date: 2018-04-23 08:21:38 +0200 (Mo., 23 Apr 2018) $
 *	Last changed by	:	$Author: b7bolm $
 *	URL				:	$URL: http://almscdc.swisslog.com/repo/SWPD/Development/BoxControlFramework/20_Release/trunk/01_Software/BCF/BCF/JumpStart/20_Product/10_App/14_Groups/10_Lib/10_Conv/01_DUTs/10_Dummy/ST_CFG_GroupManager.TcDUT $
 *
 *	Purpose			:	GroupManager configuration structure.
 *
 * ------------------------------------------------------------------------------------
 *	Copyright Swisslog [IP AG], Switzerland. All rights reserved.
 * 
 * ------------------------------------------------------------------------------------
 *	
 * 	Revision History: 
 *
 * 	VERSION			DATE			INITIALS			DESCRIPTION
 *	0.1				01.01.2001		swl					Example
 *
 **************************************************************************************)
STRUCT
	// Allocate all elements of each group
	Group	: ARRAY[G_BEGIN_GROUP..G_END_GROUP] OF ST_GroupManagerElementMember;
END_STRUCT
END_TYPE

// ---- 20_Product/10_BCF/11_Conv/11_Com/11_ITC/01_DUTs/E_ITC_MsgTypeConv.TcDUT
TYPE E_ITC_MsgTypeConv :
(**************************************************************************************
 * 	Application		:	BoxControl Framework
 *	Revision		:	$Revision: 404529 $
 *	Revision date	:	$Date: 2018-04-23 08:21:38 +0200 (Mo., 23 Apr 2018) $
 *	Last changed by	:	$Author: b7bolm $
 *	URL				:	$URL: http://almscdc.swisslog.com/repo/SWPD/Development/BoxControlFramework/20_Release/trunk/01_Software/BCF/BCF/JumpStart/20_Product/10_App/11_Com/10_Lib/10_Conv/11_ITC/01_DUTs/E_ITC_MsgTypeConv.TcDUT $
 *
 *	Purpose			:	ITC message types.
 *
 * ------------------------------------------------------------------------------------
 *	Copyright Swisslog [IP AG], Switzerland. All rights reserved.
 * 
 * ------------------------------------------------------------------------------------
 *	
 * 	Revision History: 
 *
 * 	VERSION			DATE			INITIALS			DESCRIPTION
 *	0.1				01.01.2001		swl					Example
 *
 **************************************************************************************)
(
	NO_MESSAGE_TYPE,
	ADD_TU_DATA,
	DIGITAL_INPUT_REQUEST,
	ELEMENT_CONTROL_REQUEST,
	ELEMENT_CONTROL_REPLY,
	ELEMENT_STATUS_REQUEST,
	ELEMENT_STATUS_REPORT,
	FUNCTION_CONTROL_REQUEST,
	FUNCTION_CONTROL_REPLY,
	FUNCTION_STATUS_REQUEST,
	FUNCTION_STATUS_REPORT,
	GROUP_CONTROL_REQUEST,
	GROUP_CONTROL_REPLY,
	GROUP_STATUS_REQUEST,
	GROUP_STATUS_REPORT,
	GLOBAL_VARIABLE_REQUEST,
	GLOBAL_VARIABLE_REPORT,
	IDENTIFICATION_REPORT,
	I_O_STATUS_REQUEST,
	I_O_STATUS_REPORT,
	MANUAL_CONTROL_REQUEST,
	MANUAL_CONTROL_REPORT,
	POSITION_OCCUPIED_REPORT,
	SUBSYSTEM_CONTROL_REQUEST,
	SUBSYSTEM_CONTROL_REPLY,
	SET_DIGITAL_OUTPUT,
	SEND_DIGITAL_INPUT,
	SCANNER_INFORMATION_REQUEST,
	SCANNER_INFORMATION_REPORT,
	SCANNER_NO_READ_REPORT,
	SUBSYSTEM_STATUS_REQUEST,
	SUBSYSTEM_STATUS_REPORT,
	TASK_DELETE_REQUEST,
	TASK_DELETE_REPORT,
	TRANSPORT_TASK_ASSIGNMENT,
	TRANSPORT_TASK_COMPLETE,
	TRANSPORT_TASK_REQUEST,
	TRANSPORT_UNIT_REQUEST,
	TRANSPORT_UNIT_REPORT,
	DATA_ACQUISITION_REQUEST,
	DATA_ACQUISITION_REPORT,
	GATHERED_DATA_REQUEST,
	GATHERED_DATA_REPORT,
	DATA_MESSAGE,
	E_ADD_TU_REPORT,
	E_ADD_TU_REQUEST,
	E_ERROR_REPORT,
	E_ERROR_REQUEST,
	E_REMOVE_TU_REPORT,
	E_REMOVE_TU_REQUEST,
	ROBOT_ACTION_ASSIGNMENT,
	ROBOT_ACTION_COMPLETE,
	ROBOT_ACTION_REQUEST,
	ROBOT_DELETE_REQUEST,
	ROBOT_DELETE_REPORT,
	VISUALIZATION_INFORMATION_REPORT,
	VISUALIZATION_INFORMATION_REQUEST
);
END_TYPE

// ---- 20_Product/10_BCF/11_Conv/11_Com/11_ITC/01_DUTs/ST_CFG_ITC_ManagerConv.TcDUT
TYPE ST_CFG_ITC_ManagerConv :
(**************************************************************************************
 * 	Application		:	BoxControl Framework
 *	Revision		:	$Revision: 404529 $
 *	Revision date	:	$Date: 2018-04-23 08:21:38 +0200 (Mo., 23 Apr 2018) $
 *	Last changed by	:	$Author: b7bolm $
 *	URL				:	$URL: http://almscdc.swisslog.com/repo/SWPD/Development/BoxControlFramework/20_Release/trunk/01_Software/BCF/BCF/JumpStart/20_Product/10_App/11_Com/10_Lib/10_Conv/11_ITC/01_DUTs/ST_CFG_ITC_ManagerConv.TcDUT $
 *
 *	Purpose			:	Configuration ITC
 *
 * ------------------------------------------------------------------------------------
 *	Copyright Swisslog [IP AG], Switzerland. All rights reserved.
 * 
 * ------------------------------------------------------------------------------------
 *	
 * 	Revision History: 
 *
 * 	VERSION			DATE			INITIALS			DESCRIPTION
 *	0.1				01.01.2001		swl					Example
 *
 **************************************************************************************)
STRUCT
	SDI_Limit			: INT; // Limit of used SDI signals
END_STRUCT
END_TYPE

// ---- 20_Product/10_BCF/11_Conv/11_Com/11_ITC/01_DUTs/ST_ITC_ADD_TU_DATA.TcDUT
TYPE ST_ITC_ADD_TU_DATA :
(**************************************************************************************
 * 	Application		:	BoxControl Framework
 *	Revision		:	$Revision: 404529 $
 *	Revision date	:	$Date: 2018-04-23 08:21:38 +0200 (Mo., 23 Apr 2018) $
 *	Last changed by	:	$Author: b7bolm $
 *	URL				:	$URL: http://almscdc.swisslog.com/repo/SWPD/Development/BoxControlFramework/20_Release/trunk/01_Software/BCF/BCF/JumpStart/20_Product/10_App/11_Com/10_Lib/10_Conv/11_ITC/01_DUTs/ST_ITC_ADD_TU_DATA.TcDUT $
 *
 *	Purpose			:	Add TU data to a zone
 *
 * ------------------------------------------------------------------------------------
 *	Copyright Swisslog [IP AG], Switzerland. All rights reserved.
 * 
 * ------------------------------------------------------------------------------------
 *	
 * 	Revision History: 
 *
 * 	VERSION			DATE			INITIALS			DESCRIPTION
 *	0.1				01.01.2001		swl					Example
 *
 **************************************************************************************)	
STRUCT
	eFunctionNumber	 	: E_FunctionNumber; // Number of the function 
	ZoneNumber	 		: INT; // Number of the zone  	
	TU_DataIndex		: DINT; // 6 Digit Tu Index	
END_STRUCT
END_TYPE

// ---- 20_Product/10_BCF/11_Conv/11_Com/11_ITC/01_DUTs/ST_ITC_ATQ.TcDUT
TYPE ST_ITC_ATQ :
(**************************************************************************************
 * 	Application		:	BoxControl Framework
 *	Revision		:	$Revision: 404529 $
 *	Revision date	:	$Date: 2018-04-23 08:21:38 +0200 (Mo., 23 Apr 2018) $
 *	Last changed by	:	$Author: b7bolm $
 *	URL				:	$URL: http://almscdc.swisslog.com/repo/SWPD/Development/BoxControlFramework/20_Release/trunk/01_Software/BCF/BCF/JumpStart/20_Product/11_Emu/11_Com/10_Lib/10_Conv/11_ITC/01_DUTs/ST_ITC_ATQ.TcDUT $
 *
 *	Purpose			:	ATQ Structure
 *
 * ------------------------------------------------------------------------------------
 *	Copyright Swisslog [IP AG], Switzerland. All rights reserved.
 * 
 * ------------------------------------------------------------------------------------
 *	
 * 	Revision History: 
 *
 * 	VERSION			DATE			INITIALS			DESCRIPTION
 *	0.1				01.01.2001		swl					Example
 *
 **************************************************************************************)
STRUCT
	Position			: STRING(Conveyor.POSITION_STRINGLENGTH); // SIS position name MM-000-0000-000
	Weight				: DINT; // Weight
	Length				: INT; // length
	Width				: INT; // Width
	Height				: INT; // Height
	LongSideLeading		: BOOL;
	LabelPresent		: INT; // Label present
	Label				: STRING(ConveyorEmulation.LABEL_STRING_LENGTH); // Label
END_STRUCT
END_TYPE

// ---- 20_Product/10_BCF/11_Conv/11_Com/11_ITC/01_DUTs/ST_ITC_ATR.TcDUT
TYPE ST_ITC_ATR :
(**************************************************************************************
 * 	Application		:	BoxControl Framework
 *	Revision		:	$Revision: 404529 $
 *	Revision date	:	$Date: 2018-04-23 08:21:38 +0200 (Mo., 23 Apr 2018) $
 *	Last changed by	:	$Author: b7bolm $
 *	URL				:	$URL: http://almscdc.swisslog.com/repo/SWPD/Development/BoxControlFramework/20_Release/trunk/01_Software/BCF/BCF/JumpStart/20_Product/10_App/11_Com/10_Lib/10_Conv/11_ITC/01_DUTs/ST_ITC_ATR.TcDUT $
 *
 *	Purpose			:	ATR Structure
 *
 * ------------------------------------------------------------------------------------
 *	Copyright Swisslog [IP AG], Switzerland. All rights reserved.
 * 
 * ------------------------------------------------------------------------------------
 *	
 * 	Revision History: 
 *
 * 	VERSION			DATE			INITIALS			DESCRIPTION
 *	0.1				01.01.2001		swl					Example
 *
 **************************************************************************************)
STRUCT
	Position		: STRING(Conveyor.POSITION_STRINGLENGTH); // 12 Digit SIS Location MM-GGG-EEEE-FF-Z
	ReturnCode		: E_ErrorConv; // 4 Digit error code
END_STRUCT
END_TYPE

// ---- 20_Product/10_BCF/11_Conv/11_Com/11_ITC/01_DUTs/ST_ITC_DAQ.TcDUT
TYPE ST_ITC_DAQ :
(**************************************************************************************
 * 	Application		:	BoxControl Framework
 *	Revision		:	$Revision: 404529 $
 *	Revision date	:	$Date: 2018-04-23 08:21:38 +0200 (Mo., 23 Apr 2018) $
 *	Last changed by	:	$Author: b7bolm $
 *	URL				:	$URL: http://almscdc.swisslog.com/repo/SWPD/Development/BoxControlFramework/20_Release/trunk/01_Software/BCF/BCF/JumpStart/20_Product/10_App/11_Com/10_Lib/10_Conv/11_ITC/01_DUTs/ST_ITC_DAQ.TcDUT $
 *
 *	Purpose			:	DAQ Structure 					
 *
 *
 * ------------------------------------------------------------------------------------
 *	Copyright Swisslog [IP AG], Switzerland. All rights reserved.
 * 
 * ------------------------------------------------------------------------------------
 *	
 * 	Revision History: 
 *
 * 	VERSION			DATE			INITIALS			DESCRIPTION
 *	0.1				01.01.2001		swl					Example
 *
 **************************************************************************************)	
STRUCT
	Position		: STRING(Conveyor.POSITION_STRINGLENGTH);// 12 Digit SIS Location MM-GGG-EEEE-FF-Z
	Code			: INT; // Request all= 0  Off All = 1
	NumberOfSets	: INT; // Number of Sets of dat in Telgram to me Proccessed 
	Set				: ARRAY[E_CM_Index.E_BEGIN_VARIABLE+1..E_CM_Index.E_END_VARIABLE-1] OF ST_CM_Settings; //Set Data 
END_STRUCT
END_TYPE

// ---- 20_Product/10_BCF/11_Conv/11_Com/11_ITC/01_DUTs/ST_ITC_DAR.TcDUT
TYPE ST_ITC_DAR :
(**************************************************************************************
 * 	Application		:	BoxControl Framework
 *	Revision		:	$Revision: 404529 $
 *	Revision date	:	$Date: 2018-04-23 08:21:38 +0200 (Mo., 23 Apr 2018) $
 *	Last changed by	:	$Author: b7bolm $
 *	URL				:	$URL: http://almscdc.swisslog.com/repo/SWPD/Development/BoxControlFramework/20_Release/trunk/01_Software/BCF/BCF/JumpStart/20_Product/10_App/11_Com/10_Lib/10_Conv/11_ITC/01_DUTs/ST_ITC_DAR.TcDUT $
 *
 *	Purpose			:	DAR Structure 					
 *
 *
 * ------------------------------------------------------------------------------------
 *	Copyright Swisslog [IP AG], Switzerland. All rights reserved.
 * 
 * ------------------------------------------------------------------------------------
 *	
 * 	Revision History: 
 *
 * 	VERSION			DATE			INITIALS			DESCRIPTION
 *	0.1				01.01.2001		swl					Example
 *
 **************************************************************************************)	
STRUCT
	Position		: STRING(Conveyor.POSITION_STRINGLENGTH);// 12 Digit SIS Location MM-GGG-EEEE-FF-Z
	Code			: INT;	// Request All = 0 Disable all =1 
	NumberOfSets	: INT;	//Number of Sets to Process in Telegram 
	Set				: ARRAY[E_CM_Index.E_BEGIN_VARIABLE+1..E_CM_Index.E_END_VARIABLE-1] OF ST_CM_Settings;
	SetOffset		: E_CM_Index;	// Offset of Set Number to send 
	eErrorCode		: E_ErrorConv;// 4 Digit error code
END_STRUCT
END_TYPE

// ---- 20_Product/10_BCF/11_Conv/11_Com/11_ITC/01_DUTs/ST_ITC_DIQ.TcDUT
TYPE ST_ITC_DIQ :
(**************************************************************************************
 * 	Application		:	BoxControl Framework
 *	Revision		:	$Revision: 404529 $
 *	Revision date	:	$Date: 2018-04-23 08:21:38 +0200 (Mo., 23 Apr 2018) $
 *	Last changed by	:	$Author: b7bolm $
 *	URL				:	$URL: http://almscdc.swisslog.com/repo/SWPD/Development/BoxControlFramework/20_Release/trunk/01_Software/BCF/BCF/JumpStart/20_Product/10_App/11_Com/10_Lib/10_Conv/11_ITC/01_DUTs/ST_ITC_DIQ.TcDUT $
 *
 *	Purpose			:	DIQ Structure
 *
 * ------------------------------------------------------------------------------------
 *	Copyright Swisslog [IP AG], Switzerland. All rights reserved.
 * 
 * ------------------------------------------------------------------------------------
 *	
 * 	Revision History: 
 *
 * 	VERSION			DATE			INITIALS			DESCRIPTION
 *	0.1				01.01.2001		swl					Example
 *
 **************************************************************************************)
STRUCT
;
END_STRUCT
END_TYPE

// ---- 20_Product/10_BCF/11_Conv/11_Com/11_ITC/01_DUTs/ST_ITC_ECQ.TcDUT
TYPE ST_ITC_ECQ :
(**************************************************************************************
 * 	Application		:	BoxControl Framework
 *	Revision		:	$Revision: 404529 $
 *	Revision date	:	$Date: 2018-04-23 08:21:38 +0200 (Mo., 23 Apr 2018) $
 *	Last changed by	:	$Author: b7bolm $
 *	URL				:	$URL: http://almscdc.swisslog.com/repo/SWPD/Development/BoxControlFramework/20_Release/trunk/01_Software/BCF/BCF/JumpStart/20_Product/10_App/11_Com/10_Lib/10_Conv/11_ITC/01_DUTs/ST_ITC_ECQ.TcDUT $
 *
 *	Purpose			:	Element Control Request.
 *
 * ------------------------------------------------------------------------------------
 *	Copyright Swisslog [IP AG], Switzerland. All rights reserved.
 * 
 * ------------------------------------------------------------------------------------
 *	
 * 	Revision History: 
 *
 * 	VERSION			DATE			INITIALS			DESCRIPTION
 *	0.1				01.01.2001		swl					Example
 *
 **************************************************************************************)
STRUCT
	Position	: STRING(Conveyor.POSITION_STRINGLENGTH);
	Code		: E_ITC_ElementControlCode; // Control code
	Variable	: DINT; // Control code variable
END_STRUCT
END_TYPE

// ---- 20_Product/10_BCF/11_Conv/11_Com/11_ITC/01_DUTs/ST_ITC_ECR.TcDUT
TYPE ST_ITC_ECR :
(**************************************************************************************
 * 	Application		:	BoxControl Framework
 *	Revision		:	$Revision: 404529 $
 *	Revision date	:	$Date: 2018-04-23 08:21:38 +0200 (Mo., 23 Apr 2018) $
 *	Last changed by	:	$Author: b7bolm $
 *	URL				:	$URL: http://almscdc.swisslog.com/repo/SWPD/Development/BoxControlFramework/20_Release/trunk/01_Software/BCF/BCF/JumpStart/20_Product/10_App/11_Com/10_Lib/10_Conv/11_ITC/01_DUTs/ST_ITC_ECR.TcDUT $
 *
 *	Purpose			:	ECR Structure
 *
 * ------------------------------------------------------------------------------------
 *	Copyright Swisslog [IP AG], Switzerland. All rights reserved.
 * 
 * ------------------------------------------------------------------------------------
 *	
 * 	Revision History: 
 *
 * 	VERSION			DATE			INITIALS			DESCRIPTION
 *	0.1				01.01.2001		swl					Example
 *
 **************************************************************************************)
STRUCT
	Position		: STRING(Conveyor.POSITION_STRINGLENGTH); // 12 Digit SIS Location MM-GGG-EEEE-LLL 
	Code			: INT; // 2 Digit Control code 
	Variable		: DINT; // 4 DigitControl code variable 
	ReturnCode		: E_ErrorConv; // 4 Digit return Code 
END_STRUCT
END_TYPE

// ---- 20_Product/10_BCF/11_Conv/11_Com/11_ITC/01_DUTs/ST_ITC_ERQ.TcDUT
TYPE ST_ITC_ERQ :
(**************************************************************************************
 * 	Application		:	BoxControl Framework
 *	Revision		:	$Revision: 404529 $
 *	Revision date	:	$Date: 2018-04-23 08:21:38 +0200 (Mo., 23 Apr 2018) $
 *	Last changed by	:	$Author: b7bolm $
 *	URL				:	$URL: http://almscdc.swisslog.com/repo/SWPD/Development/BoxControlFramework/20_Release/trunk/01_Software/BCF/BCF/JumpStart/20_Product/11_Emu/11_Com/10_Lib/10_Conv/11_ITC/01_DUTs/ST_ITC_ERQ.TcDUT $
 *
 *	Purpose			:	ERQ Structure
 *
 * ------------------------------------------------------------------------------------
 *	Copyright Swisslog [IP AG], Switzerland. All rights reserved.
 * 
 * ------------------------------------------------------------------------------------
 *	
 * 	Revision History: 
 *
 * 	VERSION			DATE			INITIALS			DESCRIPTION
 *	0.1				01.01.2001		swl					Example
 *
 **************************************************************************************)
STRUCT
	Position     		: STRING(Conveyor.POSITION_STRINGLENGTH); // SIS position name MM-000-0000-000
	Code				: INT; // Code
	ErrorCode			: INT; // Error code
END_STRUCT
END_TYPE

// ---- 20_Product/10_BCF/11_Conv/11_Com/11_ITC/01_DUTs/ST_ITC_ERR.TcDUT
TYPE ST_ITC_ERR :
(**************************************************************************************
 * 	Application		:	BoxControl Framework
 *	Revision		:	$Revision: 404529 $
 *	Revision date	:	$Date: 2018-04-23 08:21:38 +0200 (Mo., 23 Apr 2018) $
 *	Last changed by	:	$Author: b7bolm $
 *	URL				:	$URL: http://almscdc.swisslog.com/repo/SWPD/Development/BoxControlFramework/20_Release/trunk/01_Software/BCF/BCF/JumpStart/20_Product/10_App/11_Com/10_Lib/10_Conv/11_ITC/01_DUTs/ST_ITC_ERR.TcDUT $
 *
 *	Purpose			:	ERR Structure
 *
 * ------------------------------------------------------------------------------------
 *	Copyright Swisslog [IP AG], Switzerland. All rights reserved.
 * 
 * ------------------------------------------------------------------------------------
 *	
 * 	Revision History: 
 *
 * 	VERSION			DATE			INITIALS			DESCRIPTION
 *	0.1				01.01.2001		swl					Example
 *
 **************************************************************************************)
STRUCT
	Position		: STRING(Conveyor.POSITION_STRINGLENGTH); // 12 Digit SIS Location MM-GGG-EEEE-FF-Z
	Code			: INT; // 1 Digit error type code
	ReturnCode		: INT; // 4 Digit error code
END_STRUCT
END_TYPE

// ---- 20_Product/10_BCF/11_Conv/11_Com/11_ITC/01_DUTs/ST_ITC_ESQ.TcDUT
TYPE ST_ITC_ESQ :
(**************************************************************************************
 * 	Application		:	BoxControl Framework
 *	Revision		:	$Revision: 404529 $
 *	Revision date	:	$Date: 2018-04-23 08:21:38 +0200 (Mo., 23 Apr 2018) $
 *	Last changed by	:	$Author: b7bolm $
 *	URL				:	$URL: http://almscdc.swisslog.com/repo/SWPD/Development/BoxControlFramework/20_Release/trunk/01_Software/BCF/BCF/JumpStart/20_Product/10_App/11_Com/10_Lib/10_Conv/11_ITC/01_DUTs/ST_ITC_ESQ.TcDUT $
 *
 *	Purpose			:	Element Status Request.
 *
 * ------------------------------------------------------------------------------------
 *	Copyright Swisslog [IP AG], Switzerland. All rights reserved.
 * 
 * ------------------------------------------------------------------------------------
 *	
 * 	Revision History: 
 *
 * 	VERSION			DATE			INITIALS			DESCRIPTION
 *	0.1				01.01.2001		swl					Example
 *
 **************************************************************************************)
STRUCT
	Position	: STRING(Conveyor.POSITION_STRINGLENGTH);
END_STRUCT
END_TYPE

// ---- 20_Product/10_BCF/11_Conv/11_Com/11_ITC/01_DUTs/ST_ITC_ESR.TcDUT
TYPE ST_ITC_ESR :
(**************************************************************************************
 * 	Application		:	BoxControl Framework
 *	Revision		:	$Revision: 404529 $
 *	Revision date	:	$Date: 2018-04-23 08:21:38 +0200 (Mo., 23 Apr 2018) $
 *	Last changed by	:	$Author: b7bolm $
 *	URL				:	$URL: http://almscdc.swisslog.com/repo/SWPD/Development/BoxControlFramework/20_Release/trunk/01_Software/BCF/BCF/JumpStart/20_Product/10_App/11_Com/10_Lib/10_Conv/11_ITC/01_DUTs/ST_ITC_ESR.TcDUT $
 *
 *	Purpose			:	ESR Structure
 *
 * ------------------------------------------------------------------------------------
 *	Copyright Swisslog [IP AG], Switzerland. All rights reserved.
 * 
 * ------------------------------------------------------------------------------------
 *	
 * 	Revision History: 
 *
 * 	VERSION			DATE			INITIALS			DESCRIPTION
 *	0.1				01.01.2001		swl					Example
 *
 **************************************************************************************)
STRUCT
	Position 			: STRING(Conveyor.POSITION_STRINGLENGTH); // 12 Digit SIS Location MM-GGG-EEEE-LLL 
	State				: E_PositionState; // 1 Digit State 
	Enabled				: BOOL; // 1 Digit State 
	ErrorState			: E_ErrorState; // 1 Digit Error State 
	ErrorCode			: E_ErrorConv; // 4 Digit Return Code 
	ErrorType			: E_ErrorType; // 1 Digit Error Type 
	ErrorInformation	: STRING(System.ERROR_PARAM_STRINGLENGTH); // 5 Chars Error Information 
	Variable			: DINT; // 4 Digit Variable 
	ReturnCode			: E_ErrorConv; // 4 Digit error code
END_STRUCT
END_TYPE

// ---- 20_Product/10_BCF/11_Conv/11_Com/11_ITC/01_DUTs/ST_ITC_FCQ.TcDUT
TYPE ST_ITC_FCQ :
(**************************************************************************************
 * 	Application		:	BoxControl Framework
 *	Revision		:	$Revision: 404529 $
 *	Revision date	:	$Date: 2018-04-23 08:21:38 +0200 (Mo., 23 Apr 2018) $
 *	Last changed by	:	$Author: b7bolm $
 *	URL				:	$URL: http://almscdc.swisslog.com/repo/SWPD/Development/BoxControlFramework/20_Release/trunk/01_Software/BCF/BCF/JumpStart/20_Product/10_App/11_Com/10_Lib/10_Conv/11_ITC/01_DUTs/ST_ITC_FCQ.TcDUT $
 *
 *	Purpose			:	Element Control Request.
 *
 * ------------------------------------------------------------------------------------
 *	Copyright Swisslog [IP AG], Switzerland. All rights reserved.
 * 
 * ------------------------------------------------------------------------------------
 *	
 * 	Revision History: 
 *
 * 	VERSION			DATE			INITIALS			DESCRIPTION
 *	0.1				01.01.2001		swl					Example
 *
 **************************************************************************************)
STRUCT
	Position	: STRING(Conveyor.POSITION_STRINGLENGTH);
	Code		: E_ITC_FunctionControlCode; // ITC message code
	Variable	: DINT; // Control code variable
END_STRUCT
END_TYPE

// ---- 20_Product/10_BCF/11_Conv/11_Com/11_ITC/01_DUTs/ST_ITC_FCR.TcDUT
TYPE ST_ITC_FCR :
(**************************************************************************************
 * 	Application		:	BoxControl Framework
 *	Revision		:	$Revision: 404529 $
 *	Revision date	:	$Date: 2018-04-23 08:21:38 +0200 (Mo., 23 Apr 2018) $
 *	Last changed by	:	$Author: b7bolm $
 *	URL				:	$URL: http://almscdc.swisslog.com/repo/SWPD/Development/BoxControlFramework/20_Release/trunk/01_Software/BCF/BCF/JumpStart/20_Product/10_App/11_Com/10_Lib/10_Conv/11_ITC/01_DUTs/ST_ITC_FCR.TcDUT $
 *
 *	Purpose			:	FCR Structure
 *
 * ------------------------------------------------------------------------------------
 *	Copyright Swisslog [IP AG], Switzerland. All rights reserved.
 * 
 * ------------------------------------------------------------------------------------
 *	
 * 	Revision History: 
 *
 * 	VERSION			DATE			INITIALS			DESCRIPTION
 *	0.1				01.01.2001		swl					Example
 *
 **************************************************************************************)
STRUCT
	Position		: STRING(Conveyor.POSITION_STRINGLENGTH); // 12 Digit SIS Location MM-GGG-EEEE-LLL 
	Code			: INT; // 2 Digit Control code 
	Variable		: DINT; // 4 DigitControl code variable 
	ReturnCode		: E_ErrorConv; // 4 Digit return Code 
END_STRUCT
END_TYPE

// ---- 20_Product/10_BCF/11_Conv/11_Com/11_ITC/01_DUTs/ST_ITC_FSQ.TcDUT
TYPE ST_ITC_FSQ :
(**************************************************************************************
 * 	Application		:	BoxControl Framework
 *	Revision		:	$Revision: 404529 $
 *	Revision date	:	$Date: 2018-04-23 08:21:38 +0200 (Mo., 23 Apr 2018) $
 *	Last changed by	:	$Author: b7bolm $
 *	URL				:	$URL: http://almscdc.swisslog.com/repo/SWPD/Development/BoxControlFramework/20_Release/trunk/01_Software/BCF/BCF/JumpStart/20_Product/10_App/11_Com/10_Lib/10_Conv/11_ITC/01_DUTs/ST_ITC_FSQ.TcDUT $
 *
 *	Purpose			:	Function Status Request.
 *
 * ------------------------------------------------------------------------------------
 *	Copyright Swisslog [IP AG], Switzerland. All rights reserved.
 * 
 * ------------------------------------------------------------------------------------
 *	
 * 	Revision History: 
 *
 * 	VERSION			DATE			INITIALS			DESCRIPTION
 *	0.1				01.01.2001		swl					Example
 *
 **************************************************************************************)
STRUCT
	Position	: STRING(Conveyor.POSITION_STRINGLENGTH);
END_STRUCT
END_TYPE

// ---- 20_Product/10_BCF/11_Conv/11_Com/11_ITC/01_DUTs/ST_ITC_FSR.TcDUT
TYPE ST_ITC_FSR :
(**************************************************************************************
 * 	Application		:	BoxControl Framework
 *	Revision		:	$Revision: 404529 $
 *	Revision date	:	$Date: 2018-04-23 08:21:38 +0200 (Mo., 23 Apr 2018) $
 *	Last changed by	:	$Author: b7bolm $
 *	URL				:	$URL: http://almscdc.swisslog.com/repo/SWPD/Development/BoxControlFramework/20_Release/trunk/01_Software/BCF/BCF/JumpStart/20_Product/10_App/11_Com/10_Lib/10_Conv/11_ITC/01_DUTs/ST_ITC_FSR.TcDUT $
 *
 *	Purpose			:	FSR Structure
 *
 * ------------------------------------------------------------------------------------
 *	Copyright Swisslog [IP AG], Switzerland. All rights reserved.
 * 
 * ------------------------------------------------------------------------------------
 *	
 * 	Revision History: 
 *
 * 	VERSION			DATE			INITIALS			DESCRIPTION
 *	0.1				01.01.2001		swl					Example
 *
 **************************************************************************************)
STRUCT
	Position 			: STRING(Conveyor.POSITION_STRINGLENGTH); // 12 Digit SIS Location MM-GGG-EEEE-LLL 
	PrevFunctionNo		: STRING(Conveyor.POSITION_STRINGLENGTH); // SIS MM-GGG-EEEE-FF-Z
	NextFunctionNo		: STRING(Conveyor.POSITION_STRINGLENGTH); // SIS MM-GGG-EEEE-FF-Z
	eState				: E_PositionState; // State
	Enabled				: BOOL; // Enabled
	TransportState		: E_TransportState;
	TakeOverState		: E_TakeOverState;
	HandOverState		: E_HandOverState;
	TU_ID				: STRING(Conveyor.TU_ID_STRINGLENGTH); // 18 Digit SSID
	TU_Type				: INT; // TU Type
	AssignmentID		: UDINT; // Assignment ID
	LoadInformation		: INT; // 1 = Loaded, 0 = Not loaded
	Destination			: STRING(Conveyor.POSITION_STRINGLENGTH);
	eErrorState			: E_ErrorState; // Error State
	eErrorCode			: E_ErrorConv; // Return Code
	eErrorType			: E_ErrorType; // Error Type
	ErrorInformation	: STRING(System.ERROR_PARAM_STRINGLENGTH); // 5 Chars Error Information
	Variable			: DINT; // Variable
	eReturnCode			: E_ErrorConv; // Return code
END_STRUCT
END_TYPE

// ---- 20_Product/10_BCF/11_Conv/11_Com/11_ITC/01_DUTs/ST_ITC_GCQ.TcDUT
TYPE ST_ITC_GCQ :
(**************************************************************************************
 * 	Application		:	BoxControl Framework
 *	Revision		:	$Revision: 404529 $
 *	Revision date	:	$Date: 2018-04-23 08:21:38 +0200 (Mo., 23 Apr 2018) $
 *	Last changed by	:	$Author: b7bolm $
 *	URL				:	$URL: http://almscdc.swisslog.com/repo/SWPD/Development/BoxControlFramework/20_Release/trunk/01_Software/BCF/BCF/JumpStart/20_Product/10_App/11_Com/10_Lib/10_Conv/11_ITC/01_DUTs/ST_ITC_GCQ.TcDUT $
 *
 *	Purpose			:	Element Control Request.
 *
 * ------------------------------------------------------------------------------------
 *	Copyright Swisslog [IP AG], Switzerland. All rights reserved.
 * 
 * ------------------------------------------------------------------------------------
 *	
 * 	Revision History: 
 *
 * 	VERSION			DATE			INITIALS			DESCRIPTION
 *	0.1				01.01.2001		swl					Example
 *
 **************************************************************************************)
STRUCT
	Position	: STRING(Conveyor.POSITION_STRINGLENGTH);
	Code		: E_ITC_GroupControlCode; // Control code
	Variable	: DINT; // Control code variable
END_STRUCT
END_TYPE

// ---- 20_Product/10_BCF/11_Conv/11_Com/11_ITC/01_DUTs/ST_ITC_GCR.TcDUT
TYPE ST_ITC_GCR :
(**************************************************************************************
 * 	Application		:	BoxControl Framework
 *	Revision		:	$Revision: 404529 $
 *	Revision date	:	$Date: 2018-04-23 08:21:38 +0200 (Mo., 23 Apr 2018) $
 *	Last changed by	:	$Author: b7bolm $
 *	URL				:	$URL: http://almscdc.swisslog.com/repo/SWPD/Development/BoxControlFramework/20_Release/trunk/01_Software/BCF/BCF/JumpStart/20_Product/10_App/11_Com/10_Lib/10_Conv/11_ITC/01_DUTs/ST_ITC_GCR.TcDUT $
 *
 *	Purpose			:	GCR Structure
 *
 * ------------------------------------------------------------------------------------
 *	Copyright Swisslog [IP AG], Switzerland. All rights reserved.
 * 
 * ------------------------------------------------------------------------------------
 *	
 * 	Revision History: 
 *
 * 	VERSION			DATE			INITIALS			DESCRIPTION
 *	0.1				01.01.2001		swl					Example
 *
 **************************************************************************************)
STRUCT
	GroupName		: STRING(Conveyor.POSITION_STRINGLENGTH); // 12 Digit SIS Group Name MM-GGG-0000-000 
	Code			: INT; // 2 Digit Control code 
	Variable		: DINT; // 4 DigitControl code variable 
	ReturnCode		: E_ErrorConv; // 4 Digit Return Code 
END_STRUCT
END_TYPE

// ---- 20_Product/10_BCF/11_Conv/11_Com/11_ITC/01_DUTs/ST_ITC_GDQ.TcDUT
TYPE ST_ITC_GDQ :
(**************************************************************************************
 * 	Application		:	BoxControl Framework
 *	Revision		:	$Revision: 404529 $
 *	Revision date	:	$Date: 2018-04-23 08:21:38 +0200 (Mo., 23 Apr 2018) $
 *	Last changed by	:	$Author: b7bolm $
 *	URL				:	$URL: http://almscdc.swisslog.com/repo/SWPD/Development/BoxControlFramework/20_Release/trunk/01_Software/BCF/BCF/JumpStart/20_Product/10_App/11_Com/10_Lib/10_Conv/11_ITC/01_DUTs/ST_ITC_GDQ.TcDUT $
 *
 *	Purpose			:	Gathered Data Request Structure 					
 *
 *
 * ------------------------------------------------------------------------------------
 *	Copyright Swisslog [IP AG], Switzerland. All rights reserved.
 * 
 * ------------------------------------------------------------------------------------
 *	
 * 	Revision History: 
 *
 * 	VERSION			DATE			INITIALS			DESCRIPTION
 *	0.1				01.01.2001		swl					Example
 *
 **************************************************************************************)	
STRUCT
	Position: STRING(Conveyor.POSITION_STRINGLENGTH);// 12 Digit SIS Group Name MM-GGG-0000-000 
	Variable: STRING(System.CM_VARIABLENAME_STRINGLENGTH);// 20 AlphaNumeric Char Variable name 
END_STRUCT
END_TYPE

// ---- 20_Product/10_BCF/11_Conv/11_Com/11_ITC/01_DUTs/ST_ITC_GDR.TcDUT
TYPE ST_ITC_GDR :
(**************************************************************************************
 * 	Application		:	BoxControl Framework
 *	Revision		:	$Revision: 404529 $
 *	Revision date	:	$Date: 2018-04-23 08:21:38 +0200 (Mo., 23 Apr 2018) $
 *	Last changed by	:	$Author: b7bolm $
 *	URL				:	$URL: http://almscdc.swisslog.com/repo/SWPD/Development/BoxControlFramework/20_Release/trunk/01_Software/BCF/BCF/JumpStart/20_Product/10_App/11_Com/10_Lib/10_Conv/11_ITC/01_DUTs/ST_ITC_GDR.TcDUT $
 *
 *	Purpose			:		Gathered Data Report Structure 							
 *
 *
 * ------------------------------------------------------------------------------------
 *	Copyright Swisslog [IP AG], Switzerland. All rights reserved.
 * 
 * ------------------------------------------------------------------------------------
 *	
 * 	Revision History: 
 *
 * 	VERSION			DATE			INITIALS			DESCRIPTION
 *	0.1				01.01.2001		swl					Example
 *
 **************************************************************************************)	
STRUCT
	Position		: STRING(NAME_LENGTH);// 12 Digit SIS Group Name MM-GGG-0000-000 
	Variable		: STRING(System.CM_VARIABLENAME_STRINGLENGTH);// 20 AlphaNumeric Char Variable name 
	NumberOfSets	: INT;// 1 Digit Number of Sets  0-99
	DataSet			: ARRAY[0..System.CM_MAX_NUMBER_Of_ENTRIES] OF ST_CM_LOG; //Set Data  
	eReturnCode		: E_ErrorConv;// 4 Digit Return Code 
END_STRUCT
END_TYPE

// ---- 20_Product/10_BCF/11_Conv/12_E_Functions/01_DUTs/E_ActionState.TcDUT
TYPE E_ActionState :
(**************************************************************************************
 * 	Application		:	BoxControl Framework
 *	Revision		:	$Revision: 404529 $
 *	Revision date	:	$Date: 2018-04-23 08:21:38 +0200 (Mo., 23 Apr 2018) $
 *	Last changed by	:	$Author: b7bolm $
 *	URL				:	$URL: http://almscdc.swisslog.com/repo/SWPD/Development/BoxControlFramework/20_Release/trunk/01_Software/BCF/BCF/JumpStart/20_Product/10_App/12_E_Functions/10_Lib/10_Conv/10_Functions/01_DUTs/E_ActionState.TcDUT $
 *
 *	Purpose			:	Takeover signal state
 *
 * ------------------------------------------------------------------------------------
 *	Copyright Swisslog [IP AG], Switzerland. All rights reserved.
 * 
 * ------------------------------------------------------------------------------------
 *	
 * 	Revision History: 
 *
 * 	VERSION			DATE			INITIALS			DESCRIPTION
 *	0.1				01.01.2001		swl					Example 
 *
 **************************************************************************************)
(
	WAITFOR_INITILIZATION,
	WAITFOR_LEADING_EDGE,
	WAITFOR_TRAILING_EDGE
);
END_TYPE

// ---- 20_Product/10_BCF/11_Conv/12_E_Functions/01_DUTs/E_ActionType.TcDUT
TYPE E_ActionType :
(**************************************************************************************
 * 	Application		:	BoxControl Framework
 *	Revision		:	$Revision: 404529 $
 *	Revision date	:	$Date: 2018-04-23 08:21:38 +0200 (Mo., 23 Apr 2018) $
 *	Last changed by	:	$Author: b7bolm $
 *	URL				:	$URL: http://almscdc.swisslog.com/repo/SWPD/Development/BoxControlFramework/20_Release/trunk/01_Software/BCF/BCF/JumpStart/20_Product/10_App/12_E_Functions/10_Lib/10_Conv/10_Functions/01_DUTs/E_ActionType.TcDUT $
 *
 *	Purpose			:	Takeover signal state
 *
 * ------------------------------------------------------------------------------------
 *	Copyright Swisslog [IP AG], Switzerland. All rights reserved.
 * 
 * ------------------------------------------------------------------------------------
 *	
 * 	Revision History: 
 *
 * 	VERSION			DATE			INITIALS			DESCRIPTION
 *	0.1				01.01.2001		swl					Example 
 *
 **************************************************************************************)
(
	INPUT_ACTION,
	OUTPUT_ACTION
);
END_TYPE

// ---- 20_Product/10_BCF/11_Conv/12_E_Functions/01_DUTs/E_DriveDirection.TcDUT
TYPE E_DriveDirection :
(**************************************************************************************
 * 	Application		:	BoxControl Framework
 *	Revision		:	$Revision: 404529 $
 *	Revision date	:	$Date: 2018-04-23 08:21:38 +0200 (Mo., 23 Apr 2018) $
 *	Last changed by	:	$Author: b7bolm $
 *	URL				:	$URL: http://almscdc.swisslog.com/repo/SWPD/Development/BoxControlFramework/20_Release/trunk/01_Software/BCF/BCF/JumpStart/20_Product/10_App/12_E_Functions/10_Lib/10_Conv/10_Functions/01_DUTs/E_ActionState.TcDUT $
 *
 *	Purpose			:	Set direction sign for drive
 *
 * ------------------------------------------------------------------------------------
 *	Copyright Swisslog [IP AG], Switzerland. All rights reserved.
 * 
 * ------------------------------------------------------------------------------------
 *	
 * 	Revision History: 
 *
 * 	VERSION			DATE			INITIALS			DESCRIPTION
 *	0.1				01.01.2001		swl					Example 
 *
 **************************************************************************************)
(
	FWD := 1,
	BWD := -1
);
END_TYPE

// ---- 20_Product/10_BCF/11_Conv/12_E_Functions/01_DUTs/E_FunctionType.TcDUT
TYPE E_FunctionType :
(**************************************************************************************
 * 	Application		:	BoxControl Framework
 *	Revision		:	$Revision: 404529 $
 *	Revision date	:	$Date: 2018-04-23 08:21:38 +0200 (Mo., 23 Apr 2018) $
 *	Last changed by	:	$Author: b7bolm $
 *	URL				:	$URL: http://almscdc.swisslog.com/repo/SWPD/Development/BoxControlFramework/20_Release/trunk/01_Software/BCF/BCF/JumpStart/20_Product/10_App/12_E_Functions/10_Lib/10_Conv/01_DUTs/E_FunctionType.TcDUT $
 *
 *	Purpose			:	Function type definition
 *
 * ------------------------------------------------------------------------------------
 *	Copyright Swisslog [IP AG], Switzerland. All rights reserved.
 * 
 * ------------------------------------------------------------------------------------
 *	
 * 	Revision History: 
 *
 * 	VERSION			DATE			INITIALS			DESCRIPTION
 *	0.1				01.01.2001		swl					Example
 *
 **************************************************************************************)	
(
	NO_TYPE,
	Scanner
);
END_TYPE

// ---- 20_Product/10_BCF/11_Conv/12_E_Functions/01_DUTs/E_HandOverState.TcDUT
{attribute 'qualified_only'}
{attribute 'to_string'}
TYPE E_HandOverState:
(**************************************************************************************
 * 	Application		:	BoxControl Framework
 *	Revision		:	$Revision: 404529 $
 *	Revision date	:	$Date: 2018-04-23 08:21:38 +0200 (Mo., 23 Apr 2018) $
 *	Last changed by	:	$Author: b7bolm $
 *	URL				:	$URL: http://almscdc.swisslog.com/repo/SWPD/Development/BoxControlFramework/20_Release/trunk/01_Software/BCF/BCF/JumpStart/20_Product/10_App/12_E_Functions/10_Lib/10_Conv/10_Functions/01_DUTs/E_HandOverState.TcDUT $
 *
 *	Purpose			:	Handover states
 *
 * ------------------------------------------------------------------------------------
 *	Copyright Swisslog [IP AG], Switzerland. All rights reserved.
 * 
 * ------------------------------------------------------------------------------------
 *	
 * 	Revision History: 
 *
 * 	VERSION			DATE			INITIALS			DESCRIPTION
 *	0.1				01.01.2001		swl 				Example
 *
 **************************************************************************************)
(
	UNDEFINED			:= 0,
	IDLE				:= 1,
	READY				:= 2,
	ACTIVE				:= 3,
	STOP				:= 4,
	INTERRUPTED			:= 5,
	COMPLETE			:= 6
);
END_TYPE

// ---- 20_Product/10_BCF/11_Conv/12_E_Functions/01_DUTs/E_ITC_FunctionControlCode.TcDUT
TYPE E_ITC_FunctionControlCode :
(**************************************************************************************
 * 	Application		:	BoxControl Framework
 *	Revision		:	$Revision: 404529 $
 *	Revision date	:	$Date: 2018-04-23 08:21:38 +0200 (Mo., 23 Apr 2018) $
 *	Last changed by	:	$Author: b7bolm $
 *	URL				:	$URL: http://almscdc.swisslog.com/repo/SWPD/Development/BoxControlFramework/20_Release/trunk/01_Software/BCF/BCF/JumpStart/20_Product/10_App/12_E_Functions/10_Lib/10_Conv/01_DUTs/E_ITC_FunctionControlCode.TcDUT $
 *
 *	Purpose			:	Element function control request code
 *
 * ------------------------------------------------------------------------------------
 *	Copyright Swisslog [IP AG], Switzerland. All rights reserved.
 * 
 * ------------------------------------------------------------------------------------
 *	
 * 	Revision History: 
 *
 * 	VERSION			DATE			INITIALS			DESCRIPTION
 *	0.1				01.01.2001		swl					Example
 *
 **************************************************************************************)
(
	NO_CODE					:= 0, // No code
	RESET_ERROR 			:= 1, // Reset Error
	INITIALIZE 				:= 2, // Initialize
	ENABLE 					:= 4, // Enable / Disable
	SET_VARIABLE 			:= 5, // Set Variable
	SET_ERROR 				:= 20 // Set Error
);
END_TYPE

// ---- 20_Product/10_BCF/11_Conv/12_E_Functions/01_DUTs/E_Signalstate.TcDUT
TYPE E_Signalstate :
(**************************************************************************************
 * 	Application		:	BoxControl Framework
 *	Revision		:	$Revision: 404529 $
 *	Revision date	:	$Date: 2018-04-23 08:21:38 +0200 (Mo., 23 Apr 2018) $
 *	Last changed by	:	$Author: b7bolm $
 *	URL				:	$URL: http://almscdc.swisslog.com/repo/SWPD/Development/BoxControlFramework/20_Release/trunk/01_Software/BCF/BCF/JumpStart/20_Product/10_App/12_E_Functions/10_Lib/10_Conv/10_Functions/01_DUTs/E_Signalstate.TcDUT $
 *
 *	Purpose			:	Signal states
 *
 * ------------------------------------------------------------------------------------
 *	Copyright Swisslog [IP AG], Switzerland. All rights reserved.
 * 
 * ------------------------------------------------------------------------------------
 *	
 * 	Revision History: 
 *
 * 	VERSION			DATE			INITIALS			DESCRIPTION
 *	0.1				01.01.2001		swl	 				Example 
 *
 **************************************************************************************)
(
	UNKNOWN_SIGNALSTATE,
	INPUT_OFF,
	POSITIVE_EDGE,
	NEGATIVE_EDGE,
	INPUT_ON
);
END_TYPE

// ---- 20_Product/10_BCF/11_Conv/12_E_Functions/01_DUTs/E_SpeedControlState.TcDUT
{attribute 'qualified_only'}
{attribute 'strict'}
TYPE E_SpeedControlState :
(
	STOPPED,
	ACCELERATE,
	RUNNING,
	DECELERATE
);
END_TYPE

// ---- 20_Product/10_BCF/11_Conv/12_E_Functions/01_DUTs/E_TakeoverSignalstate.TcDUT
TYPE E_TakeoverSignalstate :
(**************************************************************************************
 * 	Application		:	BoxControl Framework
 *	Revision		:	$Revision: 404529 $
 *	Revision date	:	$Date: 2018-04-23 08:21:38 +0200 (Mo., 23 Apr 2018) $
 *	Last changed by	:	$Author: b7bolm $
 *	URL				:	$URL: http://almscdc.swisslog.com/repo/SWPD/Development/BoxControlFramework/20_Release/trunk/01_Software/BCF/BCF/JumpStart/20_Product/10_App/12_E_Functions/10_Lib/10_Conv/10_Functions/01_DUTs/E_TakeoverSignalstate.TcDUT $
 *
 *	Purpose			:	Takeover signal state
 *
 * ------------------------------------------------------------------------------------
 *	Copyright Swisslog [IP AG], Switzerland. All rights reserved.
 * 
 * ------------------------------------------------------------------------------------
 *	
 * 	Revision History: 
 *
 * 	VERSION			DATE			INITIALS			DESCRIPTION
 *	0.1				01.01.2001		swl					Example 
 *
 **************************************************************************************)
(
	WAITFOR_INITILIZATION,
	WAITFOR_LEADING_EDGE,
	WAITFOR_TRAILING_EDGE
);
END_TYPE

// ---- 20_Product/10_BCF/11_Conv/12_E_Functions/01_DUTs/E_TakeOverState.TcDUT
{attribute 'qualified_only'}
{attribute 'to_string'}
TYPE E_TakeOverState:
(**************************************************************************************
 * 	Application		:	BoxControl Framework
 *	Revision		:	$Revision: 404529 $
 *	Revision date	:	$Date: 2018-04-23 08:21:38 +0200 (Mo., 23 Apr 2018) $
 *	Last changed by	:	$Author: b7bolm $
 *	URL				:	$URL: http://almscdc.swisslog.com/repo/SWPD/Development/BoxControlFramework/20_Release/trunk/01_Software/BCF/BCF/JumpStart/20_Product/10_App/12_E_Functions/10_Lib/10_Conv/10_Functions/01_DUTs/E_TakeOverState.TcDUT $
 *
 *	Purpose			:	TakeOver states
 *
 * ------------------------------------------------------------------------------------
 *	Copyright Swisslog [IP AG], Switzerland. All rights reserved.
 * 
 * ------------------------------------------------------------------------------------
 *	
 * 	Revision History: 
 *
 * 	VERSION			DATE			INITIALS			DESCRIPTION
 *	0.1				01.01.2001		swl					Example 
 *
 **************************************************************************************)
(
	UNDEFINED			:= 0,
	IDLE				:= 1,
	READY				:= 2,
	ACTIVE				:= 4,
	STOP				:= 5,
	INTERRUPTED			:= 6,
	COMPLETE			:= 7
);
END_TYPE

// ---- 20_Product/10_BCF/11_Conv/12_E_Functions/01_DUTs/E_TransportState.TcDUT
{attribute 'qualified_only'}
{attribute 'to_string'}
{attribute 'strict'}
TYPE E_TransportState:
(**************************************************************************************
 * 	Application		:	BoxControl Framework
 *	Revision		:	$Revision: 404529 $
 *	Revision date	:	$Date: 2018-04-23 08:21:38 +0200 (Mo., 23 Apr 2018) $
 *	Last changed by	:	$Author: b7bolm $
 *	URL				:	$URL: http://almscdc.swisslog.com/repo/SWPD/Development/BoxControlFramework/20_Release/trunk/01_Software/BCF/BCF/JumpStart/20_Product/10_App/12_E_Functions/10_Lib/10_Conv/10_Functions/01_DUTs/E_TransportState.TcDUT $
 *
 *	Purpose			:	Transport states
 *
 * ------------------------------------------------------------------------------------
 *	Copyright Swisslog [IP AG], Switzerland. All rights reserved.
 * 
 * ------------------------------------------------------------------------------------
 *	
 * 	Revision History: 
 *
 * 	VERSION			DATE			INITIALS			DESCRIPTION
 *	0.1				01.01.2001		swl					Example
 *
 **************************************************************************************)
(
	UNDEFINED			:= 0,
	IDLE				:= 1,
	FREE_RUN			:= 2,
	FREE				:= 3,
	TAKEOVER			:= 4,
	OCCUPIED			:= 5,
	HANDOVER			:= 6,
	CLEARING			:= 7,
	FEEDIN				:= 8,
	FEEDIN_STOP			:= 9,
	MULTIZONE			:= 10,
	MULTIZONE_OCCUPIED	:= 11,
	MULTIZONE_STOP		:= 12,
	FEED_FW				:= 13,
	MULTI_TU			:= 14,
	MULTI_TU_OCCUPIED	:= 15,
	MULTI_TU_STOP		:= 16,
	SIMULTANEOUS		:= 17,
	SIMULTANEOUS_OCCUPIED := 18,
	SIMULTANEOUS_STOP	:= 19
);
END_TYPE

// ---- 20_Product/10_BCF/11_Conv/12_E_Functions/01_DUTs/E_TUR_SendModes.TcDUT
{attribute 'qualified_only'}
{attribute 'strict'}
TYPE E_TUR_SendModes:
	(**************************************************************************************
 * 	Application		:	BoxControl Framework
 *	Revision		:	$Revision: 465637 $
 *	Revision date	:	$Date: 2020-11-13 12:51:08 +0100 (fre, 13 nov 2020) $
 *	Last changed by	:	$Author: b7lipim $
 *	URL				:	$URL: http://almscdc.swisslog.com/repo/SWPD/Development/BoxControlFramework/20_Release/tags/R1.12.0/01_Software/BCF/BCF/JumpStart/20_Product/10_BCF/11_Conv/12_E_Functions/01_DUTs/E_TUR_SendModes.TcDUT $
 *
 *
 *	Purpose			:	Additional control over when the TUR is sent if requested on TU data index deletion of the zone.
 *
 * ------------------------------------------------------------------------------------
 *	Copyright Swisslog [IP AG], Switzerland. All rights reserved.
 * 
 * ------------------------------------------------------------------------------------
 *	
 * 	Revision History: 
 *
 * 	VERSION			DATE			INITIALS			DESCRIPTION
 *	0.1				15.07.2020		jmu					First version
 *
 **************************************************************************************)
(
	ALWAYS								:= 0,	// always sent on data index deletion if requested
	DISABLED							:= 1,	// never sent on data index deletion, even if requested
	DISABLE_ON_UNKNOWN_ASSIGNMENT		:= 2,	// not sent on data index deletion if assignment is unknown
	DISABLE_ON_UNKNOWN_TU				:= 3,	// not sent on data index deletion if TU-id is unknown
	DISABLE_ON_UNKNOWN_TU_ASSIGNMENT	:= 4	// not sent on data index deletion if assignment or TU-id is unknown
) := ALWAYS;
END_TYPE

// ---- 20_Product/10_BCF/11_Conv/12_E_Functions/01_DUTs/ST_AddOn.TcDUT
TYPE ST_AddOn :
(**************************************************************************************
 * 	Application		:	BoxControl Framework
 *	Revision		:	$Revision: 404529 $
 *	Revision date	:	$Date: 2018-04-23 08:21:38 +0200 (Mo., 23 Apr 2018) $
 *	Last changed by	:	$Author: b7bolm $
 *	URL				:	$URL: http://almscdc.swisslog.com/repo/SWPD/Development/BoxControlFramework/20_Release/trunk/01_Software/BCF/BCF/JumpStart/20_Product/10_App/12_E_Functions/10_Lib/10_Conv/01_DUTs/ST_AddOn.TcDUT $
 *
 *	Purpose			:	AddOn structure
 *
 * ------------------------------------------------------------------------------------
 *	Copyright Swisslog [IP AG], Switzerland. All rights reserved.
 * 
 * ------------------------------------------------------------------------------------
 *	
 * 	Revision History: 
 *
 * 	VERSION			DATE			INITIALS			DESCRIPTION
 *	0.1				01.01.2001		swl					Example
 *
 **************************************************************************************)
STRUCT
	eFunctionNumber		: E_FunctionNumber; // Function number
	ZoneNumber			: INT; // Zone number
	eFunctionType		: E_FunctionType; // Function type
	Orders				: ST_AddOnOrders; // Orders
END_STRUCT
END_TYPE

// ---- 20_Product/10_BCF/11_Conv/12_E_Functions/01_DUTs/ST_AddOnData.TcDUT
TYPE ST_AddOnData :
(**************************************************************************************
 * 	Application		:	BoxControl Framework
 *	Revision		:	$Revision: 404529 $
 *	Revision date	:	$Date: 2018-04-23 08:21:38 +0200 (Mo., 23 Apr 2018) $
 *	Last changed by	:	$Author: b7bolm $
 *	URL				:	$URL: http://almscdc.swisslog.com/repo/SWPD/Development/BoxControlFramework/20_Release/trunk/01_Software/BCF/BCF/JumpStart/20_Product/10_App/12_E_Functions/10_Lib/10_Conv/01_DUTs/ST_AddOnData.TcDUT $
 *
 *	Purpose			:	Internal addon data
 *
 * ------------------------------------------------------------------------------------
 *	Copyright Swisslog [IP AG], Switzerland. All rights reserved.
 * 
 * ------------------------------------------------------------------------------------
 *	
 * 	Revision History: 
 *
 * 	VERSION			DATE			INITIALS			DESCRIPTION
 *	0.1				01.01.2001		swl					Example
 *
 **************************************************************************************)
STRUCT
	Counter		: ARRAY[1..5] OF DINT; // Various counter
	LastTU_ID	: STRING(Conveyor.TU_ID_STRINGLENGTH); // Last Tu ID
END_STRUCT
END_TYPE

// ---- 20_Product/10_BCF/11_Conv/12_E_Functions/01_DUTs/ST_AddonEntry.TcDUT
TYPE ST_AddonEntry :
(**************************************************************************************
 * 	Application		:	BoxControl Framework
 *	Revision		:	$Revision: 404529 $
 *	Revision date	:	$Date: 2018-04-23 08:21:38 +0200 (Mo., 23 Apr 2018) $
 *	Last changed by	:	$Author: b7bolm $
 *	URL				:	$URL: http://almscdc.swisslog.com/repo/SWPD/Development/BoxControlFramework/20_Release/trunk/01_Software/BCF/BCF/JumpStart/20_Product/10_App/12_E_Functions/10_Lib/10_Conv/01_DUTs/ST_AddonEntry.TcDUT $
 *
 *	Purpose			:	Function Addon entry
 *
 * ------------------------------------------------------------------------------------
 *	Copyright Swisslog [IP AG], Switzerland. All rights reserved.
 * 
 * ------------------------------------------------------------------------------------
 *	
 * 	Revision History: 
 *
 * 	VERSION			DATE			INITIALS			DESCRIPTION
 *	0.1				01.01.2001		swl					Example
 *
 **************************************************************************************)
STRUCT
	eFunctionNumber		: E_FunctionNumber; // Function number
	ZoneNumber			: INT; // Zone number
END_STRUCT
END_TYPE

// ---- 20_Product/10_BCF/11_Conv/12_E_Functions/01_DUTs/ST_AddOnOrders.TcDUT
TYPE ST_AddOnOrders :
(**************************************************************************************
 * 	Application		:	BoxControl Framework
 *	Revision		:	$Revision: 474969 $
 *	Revision date	:	$Date: 2021-04-08 19:53:18 +0200 (tor, 08 apr 2021) $
 *	Last changed by	:	$Author: d7mangc $
 *	URL				:	$URL: http://almscdc.swisslog.com/repo/SWPD/Development/BoxControlFramework/20_Release/tags/R1.12.0/01_Software/BCF/BCF/JumpStart/20_Product/10_BCF/11_Conv/12_E_Functions/01_DUTs/ST_AddOnOrders.TcDUT $
 *
 *	Purpose			:	AddOn orders (output)
 *
 * ------------------------------------------------------------------------------------
 *	Copyright Swisslog [IP AG], Switzerland. All rights reserved.
 * 
 * ------------------------------------------------------------------------------------
 *	
 * 	Revision History: 
 *
 *  VERSION DATE         INITIALS     DESCRIPTION
 *  0.0     DD.MM.YYYY   (name)       (explain customized modifications)
 *
 **************************************************************************************)
STRUCT
  Enable                		: BOOL; // General enable
  EnableTakeover        		: BOOL; // Enable takeover
  EnableHandover        		: BOOL; // Enable handover
  EnableSimultaneousTransport 	: BOOL; // Enable simultaneous transport mode
  DataReady             		: BOOL; // Process of add-on function is complete
  DataValid             		: BOOL; // Scanner specific - data valid
  TU_DataIndex                	: DINT; // TU data index
  AddOnSensor                 	: BOOL; // Used when zone is configured to use AddOn sensor if not UseOwnSensor
  UseOwnSensor                	: BOOL; // AddOn forces the use of the own sensor instead of the addonsensor
  AllowDriveTakeover            : BOOL; // Used to sync the driving motors when slugging
  AllowDriveHandover            : BOOL; // Used to sync the driving motors when slugging
END_STRUCT
END_TYPE

// ---- 20_Product/10_BCF/11_Conv/12_E_Functions/01_DUTs/ST_AddOnResult.TcDUT
TYPE ST_AddOnResult :
(**************************************************************************************
 * 	Application		:	BoxControl Framework
 *	Revision		:	$Revision: 404529 $
 *	Revision date	:	$Date: 2018-04-23 08:21:38 +0200 (Mo., 23 Apr 2018) $
 *	Last changed by	:	$Author: b7bolm $
 *	URL				:	$URL: http://almscdc.swisslog.com/repo/SWPD/Development/BoxControlFramework/20_Release/trunk/01_Software/BCF/BCF/JumpStart/20_Product/10_App/12_E_Functions/10_Lib/10_Conv/01_DUTs/ST_AddOnResult.TcDUT $
 *
 *	Purpose			:	AddOn result structure
 *
 * ------------------------------------------------------------------------------------
 *	Copyright Swisslog [IP AG], Switzerland. All rights reserved.
 * 
 * ------------------------------------------------------------------------------------
 *	
 * 	Revision History: 
 *
 * 	VERSION			DATE			INITIALS			DESCRIPTION
 *	0.1				01.01.2001		swl					Example
 *
 **************************************************************************************)
STRUCT
	NoAddons			: BOOL; // No addons
	Orders				: ST_AddOnOrders; // Orders
END_STRUCT
END_TYPE

// ---- 20_Product/10_BCF/11_Conv/12_E_Functions/01_DUTs/ST_CFG_Function.TcDUT
TYPE ST_CFG_Function :
(**************************************************************************************
 * 	Application		:	BoxControl Framework
 *	Revision		:	$Revision: 404529 $
 *	Revision date	:	$Date: 2018-04-23 08:21:38 +0200 (Mo., 23 Apr 2018) $
 *	Last changed by	:	$Author: b7bolm $
 *	URL				:	$URL: http://almscdc.swisslog.com/repo/SWPD/Development/BoxControlFramework/20_Release/trunk/01_Software/BCF/BCF/JumpStart/20_Product/10_App/12_E_Functions/10_Lib/10_Conv/01_DUTs/10_Dummy/ST_CFG_Function.TcDUT $
 *
 *	Purpose			:	Base function config
 *
 * ------------------------------------------------------------------------------------
 *	Copyright Swisslog [IP AG], Switzerland. All rights reserved.
 * 
 * ------------------------------------------------------------------------------------
 *	
 * 	Revision History: 
 *
 * 	VERSION			DATE			INITIALS			DESCRIPTION
 *	0.1				01.01.2001		swl					Example
 *
 **************************************************************************************)
STRUCT
	FunctionName					: STRING(NAME_LENGTH); // Name of the function
	eFunctionNumber					: E_FunctionNumber; // Number oft the function
	eFunctionType					: E_FunctionType; // Function type
	NumberOfZones					: INT; // Number of zones
	eElementLink					: E_ElementNumber; // Link to element (mandatory)
	FunctionLink					: ST_CFG_FunctionLink; // Link to other element function (option)
	eAdjacentFunctionNumberSide 	: ARRAY [1..4] OF E_FunctionNumber; // Adjacent function number
	ePrevFunctionNumber				: E_FunctionNumber; // Previous function number
	eNextFunctionNumber				: E_FunctionNumber; // Next function number
	eExternalSTI_FunctionNumber		: ARRAY [1..Conveyor.NUMBER_OF_STI] OF E_FunctionNumber; // External Subsystem interface numbers		
	FlowDirectionREV    			: BOOL; // Flow direction reverse
	Zone							: ARRAY [1..NUMBER_OF_ZONES_PER_FUNCTION] OF ST_CFG_Zone;
	Axis_Orientation				: E_Axis_Orientation; // Orientation of function axis on element
	Acceleration					: INT; // Acceleration [mm/s^2]		
END_STRUCT
END_TYPE

// ---- 20_Product/10_BCF/11_Conv/12_E_Functions/01_DUTs/ST_CFG_FunctionLink.TcDUT
TYPE ST_CFG_FunctionLink :
(**************************************************************************************
 * 	Application		:	BoxControl Framework
 *	Revision		:	$Revision: 404529 $
 *	Revision date	:	$Date: 2018-04-23 08:21:38 +0200 (Mo., 23 Apr 2018) $
 *	Last changed by	:	$Author: b7bolm $
 *	URL				:	$URL: http://almscdc.swisslog.com/repo/SWPD/Development/BoxControlFramework/20_Release/trunk/01_Software/BCF/BCF/JumpStart/20_Product/10_App/12_E_Functions/10_Lib/10_Conv/01_DUTs/10_Dummy/ST_CFG_FunctionLink.TcDUT $
 *
 *	Purpose			:	Function link config
 *
 * ------------------------------------------------------------------------------------
 *	Copyright Swisslog [IP AG], Switzerland. All rights reserved.
 * 
 * ------------------------------------------------------------------------------------
 *	
 * 	Revision History: 
 *
 * 	VERSION			DATE			INITIALS			DESCRIPTION
 *	0.1				01.01.2001		swl					Example
 *
 **************************************************************************************)
STRUCT
	eFunctionNumber		: E_FunctionNumber; // Number of the function 
	ZoneNumber			: INT; // Number of the zone in the function 
END_STRUCT
END_TYPE

